KUKA KRL program: MyProgram_019().src

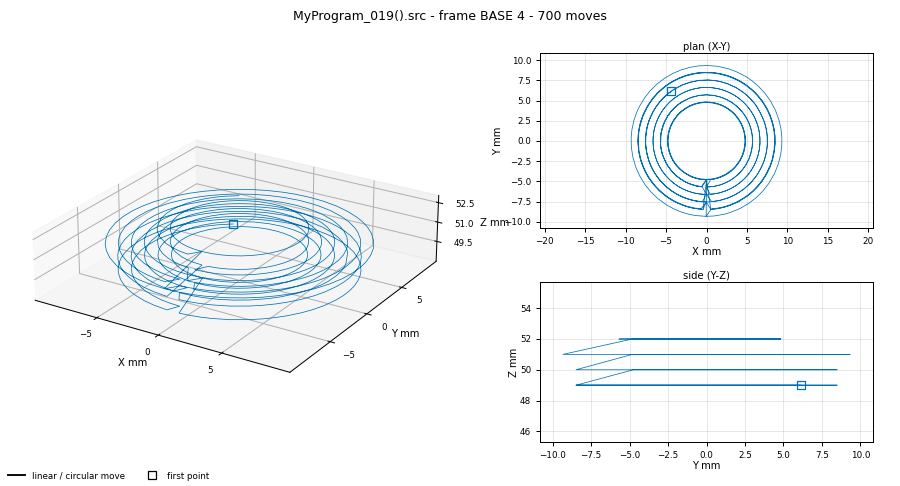
[picture p0: tool path of MyProgram_019().src in frame BASE 4, 700 of 700 moves have a stored position in this frame; points joined in program order, loops and branches not executed]
&ACCESS RVP
&REL 1
&PARAM TEMPLATE = C:\KRC\Roboter\Template\vorgabe
&PARAM EDITMASK = *
DEF MyProgram_019()
; ---- Setting reference (Base) ----
$BASE = BASE_DATA[4]

; --------------------------
; ---- Setting tool (TCP) ----
$TOOL = TOOL_DATA[3]
; --------------------------

$VEL.CP = VEL_APROX_PRINT
Startdeposition()
$VEL.CP = VEL_PRINT
LIN {X -4.3861,Y 6.1542,Z 49,A -2.5539,B 0,C 0,E1 0.1598,E2 90.072} C_DIS
LIN {X -5.2131,Y 5.4702,Z 49,A -2.6133,B 0,C 0,E1 0.1598,E2 90.0718} C_DIS
LIN {X -5.8474,Y 4.7889,Z 49,A -2.6655,B 0,C 0,E1 0.1598,E2 90.0718} C_DIS
LIN {X -6.5348,Y 3.7984,Z 49,A -2.7326,B 0,C 0,E1 0.1598,E2 90.0714} C_DIS
LIN {X -7.1278,Y 2.5114,Z 49,A -2.8086,B 0,C 0,E1 0.1598,E2 90.071} C_DIS
LIN {X -7.4027,Y 1.5183,Z 49,A -2.861,B 0,C 0,E1 0.1598,E2 90.0712} C_DIS
LIN {X -7.5273,Y 0.6846,Z 49,A -2.9011,B 0,C 0,E1 0.1598,E2 90.0714} C_DIS
LIN {X -7.5434,Y -0.4544,Z 49,A -2.9495,B 0,C 0,E1 0.1598,E2 90.0709} C_DIS
LIN {X -7.4365,Y -1.3517,Z 49,A -2.9839,B 0,C 0,E1 0.1598,E2 90.0712} C_DIS
LIN {X -7.1354,Y -2.475,Z 49,A -3.0202,B 0,C 0,E1 0.1598,E2 90.0709} C_DIS
LIN {X -6.8384,Y -3.2059,Z 49,A -3.0406,B 0,C 0,E1 0.1598,E2 90.0712} C_DIS
LIN {X -6.4681,Y -3.9026,Z 49,A -3.0566,B 0,C 0,E1 0.1598,E2 90.0712} C_DIS
LIN {X -5.8075,Y -4.8355,Z 49,A -3.0718,B 0,C 0,E1 0.1598,E2 90.071} C_DIS
LIN {X -5.1034,Y -5.5744,Z 49,A -3.0774,B 0,C 0,E1 0.1598,E2 90.0711} C_DIS
LIN {X -4.3813,Y -6.1518,Z 49,A -3.0756,B 0,C 0,E1 0.1598,E2 90.0713} C_DIS
LIN {X -3.5989,Y -6.6446,Z 49,A -3.0679,B 0,C 0,E1 0.1598,E2 90.0713} C_DIS
LIN {X -2.6446,Y -7.0747,Z 49,A -3.0512,B 0,C 0,E1 0.1598,E2 90.0713} C_DIS
LIN {X -1.6257,Y -7.3802,Z 49,A -3.0269,B 0,C 0,E1 0.1598,E2 90.0715} C_DIS
LIN {X -0.8328,Y -7.5076,Z 49,A -3.0033,B 0,C 0,E1 0.1598,E2 90.0715} C_DIS
LIN {X -0.0313,Y -7.5551,Z 49,A -2.976,B 0,C 0,E1 0.1598,E2 90.0716} C_DIS
Enddeposition()
LIN {X -0.0313,Y -7.5551,Z 49,A -2.976,B 0,C 0,E1 0.1598,E2 90.0716} C_DIS
Startdeposition()
$VEL.CP = VEL_PRINT
LIN {X -0.4344,Y -8.4805,Z 49,A -3.0298,B 0,C 0,E1 0.1598,E2 90.071} C_DIS
LIN {X -1.5865,Y -8.3368,Z 49,A -3.0665,B 0,C 0,E1 0.1598,E2 90.0714} C_DIS
LIN {X -2.5442,Y -8.1001,Z 49,A -3.0915,B 0,C 0,E1 0.1598,E2 90.0714} C_DIS
LIN {X -3.6406,Y -7.6652,Z 49,A -3.1131,B 0,C 0,E1 0.1598,E2 90.0713} C_DIS
LIN {X -4.3696,Y -7.2748,Z 49,A -3.1232,B 0,C 0,E1 0.1598,E2 90.0713} C_DIS
LIN {X -5.0572,Y -6.8153,Z 49,A -3.1289,B 0,C 0,E1 0.1598,E2 90.0713} C_DIS
LIN {X -5.8504,Y -6.1524,Z 49,A -3.1297,B 0,C 0,E1 0.1598,E2 90.0711} C_DIS
LIN {X -6.6291,Y -5.2974,Z 49,A -3.1218,B 0,C 0,E1 0.1598,E2 90.071} C_DIS
LIN {X -7.1233,Y -4.6123,Z 49,A -3.111,B 0,C 0,E1 0.1598,E2 90.0712} C_DIS
LIN {X -7.547,Y -3.8813,Z 49,A -3.0955,B 0,C 0,E1 0.1598,E2 90.0712} C_DIS
LIN {X -7.8959,Y -3.1119,Z 49,A -3.0757,B 0,C 0,E1 0.1598,E2 90.0712} C_DIS
LIN {X -8.1665,Y -2.3115,Z 49,A -3.0517,B 0,C 0,E1 0.1598,E2 90.0712} C_DIS
LIN {X -8.3936,Y -1.2801,Z 49,A -3.0161,B 0,C 0,E1 0.1598,E2 90.0709} C_DIS
LIN {X -8.487,Y -0.0694,Z 49,A -2.9681,B 0,C 0,E1 0.1598,E2 90.0709} C_DIS
LIN {X -8.4542,Y 0.7473,Z 49,A -2.9327,B 0,C 0,E1 0.1598,E2 90.0713} C_DIS
LIN {X -8.3422,Y 1.5569,Z 49,A -2.8944,B 0,C 0,E1 0.1598,E2 90.0713} C_DIS
LIN {X -8.154,Y 2.3523,Z 49,A -2.8538,B 0,C 0,E1 0.1598,E2 90.0714} C_DIS
LIN {X -7.8156,Y 3.3164,Z 49,A -2.8003,B 0,C 0,E1 0.1598,E2 90.0713} C_DIS
LIN {X -7.2981,Y 4.3333,Z 49,A -2.7381,B 0,C 0,E1 0.1598,E2 90.0713} C_DIS
LIN {X -6.6452,Y 5.2858,Z 49,A -2.6739,B 0,C 0,E1 0.1598,E2 90.0716} C_DIS
LIN {X -5.9556,Y 6.045,Z 49,A -2.6165,B 0,C 0,E1 0.1598,E2 90.0718} C_DIS
LIN {X -5.3443,Y 6.5923,Z 49,A -2.5709,B 0,C 0,E1 0.1598,E2 90.072} C_DIS
LIN {X -4.5122,Y 7.192,Z 49,A -2.5148,B 0,C 0,E1 0.1598,E2 90.072} C_DIS
LIN {X -3.4136,Y 7.7681,Z 49,A -2.4499,B 0,C 0,E1 0.1598,E2 90.0721} C_DIS
LIN {X -2.6211,Y 8.0702,Z 49,A -2.4079,B 0,C 0,E1 0.1598,E2 90.0723} C_DIS
LIN {X -1.8024,Y 8.2917,Z 49,A -2.3683,B 0,C 0,E1 0.1598,E2 90.0723} C_DIS
LIN {X -0.9657,Y 8.4308,Z 49,A -2.3315,B 0,C 0,E1 0.1598,E2 90.0725} C_DIS
LIN {X -0.1194,Y 8.4866,Z 49,A -2.2979,B 0,C 0,E1 0.1598,E2 90.0725} C_DIS
LIN {X 0.7283,Y 8.4556,Z 49,A -2.2679,B 0,C 0,E1 0.1598,E2 90.0725} C_DIS
LIN {X 1.5686,Y 8.3401,Z 49,A -2.2418,B 0,C 0,E1 0.1598,E2 90.0725} C_DIS
LIN {X 2.3934,Y 8.1418,Z 49,A -2.2198,B 0,C 0,E1 0.1598,E2 90.0725} C_DIS
LIN {X 3.1943,Y 7.8623,Z 49,A -2.2021,B 0,C 0,E1 0.1598,E2 90.0725} C_DIS
LIN {X 3.9633,Y 7.5043,Z 49,A -2.1889,B 0,C 0,E1 0.1598,E2 90.0725} C_DIS
LIN {X 4.6928,Y 7.0713,Z 49,A -2.1804,B 0,C 0,E1 0.1598,E2 90.0725} C_DIS
LIN {X 5.5399,Y 6.4335,Z 49,A -2.1761,B 0,C 0,E1 0.1598,E2 90.0724} C_DIS
LIN {X 6.4322,Y 5.5394,Z 49,A -2.1811,B 0,C 0,E1 0.1598,E2 90.0721} C_DIS
LIN {X 6.9258,Y 4.9117,Z 49,A -2.1898,B 0,C 0,E1 0.1598,E2 90.0723} C_DIS
LIN {X 7.4984,Y 3.9766,Z 49,A -2.2084,B 0,C 0,E1 0.1598,E2 90.0721} C_DIS
LIN {X 7.8686,Y 3.1812,Z 49,A -2.2288,B 0,C 0,E1 0.1598,E2 90.0722} C_DIS
LIN {X 8.1545,Y 2.3518,Z 49,A -2.2537,B 0,C 0,E1 0.1598,E2 90.0722} C_DIS
LIN {X 8.3544,Y 1.4976,Z 49,A -2.2828,B 0,C 0,E1 0.1598,E2 90.0721} C_DIS
LIN {X 8.4655,Y 0.6273,Z 49,A -2.3159,B 0,C 0,E1 0.1598,E2 90.0721} C_DIS
LIN {X 8.4847,Y -0.2497,Z 49,A -2.3526,B 0,C 0,E1 0.1598,E2 90.072} C_DIS
LIN {X 8.4122,Y -1.1239,Z 49,A -2.3927,B 0,C 0,E1 0.1598,E2 90.072} C_DIS
LIN {X 8.1761,Y -2.2938,Z 49,A -2.4511,B 0,C 0,E1 0.1598,E2 90.0716} C_DIS
LIN {X 7.8313,Y -3.2796,Z 49,A -2.506,B 0,C 0,E1 0.1598,E2 90.0716} C_DIS
LIN {X 7.4497,Y -4.0724,Z 49,A -2.5541,B 0,C 0,E1 0.1598,E2 90.0718} C_DIS
LIN {X 6.8636,Y -4.9906,Z 49,A -2.6148,B 0,C 0,E1 0.1598,E2 90.0717} C_DIS
LIN {X 6.3158,Y -5.6683,Z 49,A -2.6641,B 0,C 0,E1 0.1598,E2 90.0717} C_DIS
LIN {X 5.7013,Y -6.2863,Z 49,A -2.7131,B 0,C 0,E1 0.1598,E2 90.0717} C_DIS
LIN {X 5.0268,Y -6.8381,Z 49,A -2.7614,B 0,C 0,E1 0.1598,E2 90.0717} C_DIS
LIN {X 3.9381,Y -7.5235,Z 49,A -2.8305,B 0,C 0,E1 0.1598,E2 90.0716} C_DIS
LIN {X 2.8026,Y -8.0106,Z 49,A -2.8931,B 0,C 0,E1 0.1598,E2 90.0716} C_DIS
LIN {X 2.0583,Y -8.2323,Z 49,A -2.9299,B 0,C 0,E1 0.1598,E2 90.0716} C_DIS
LIN {X 1.2972,Y -8.386,Z 49,A -2.9643,B 0,C 0,E1 0.1598,E2 90.0716} C_DIS
LIN {X 0.5254,Y -8.4707,Z 49,A -2.9962,B 0,C 0,E1 0.1598,E2 90.0716} C_DIS
LIN {X 0.5254,Y -8.4707,Z 49,A -2.9962,B 0,C 0,E1 0.1598,E2 90.0716} C_DIS
Enddeposition()
LIN {X 0.0009,Y -4.7523,Z 50,A -2.8426,B 0,C 0,E1 0.1598,E2 90.0604} C_DIS
Startdeposition()
$VEL.CP = VEL_PRINT
LIN {X 0.0009,Y -4.7523,Z 50,A -2.8483,B 0,C 0,E1 0.1598,E2 90.0661} C_DIS
LIN {X 0.8085,Y -4.6841,Z 50,A -2.8207,B 0,C 0,E1 0.1598,E2 90.0711} C_DIS
LIN {X 1.4382,Y -4.5283,Z 50,A -2.7915,B 0,C 0,E1 0.1598,E2 90.0718} C_DIS
LIN {X 2.3301,Y -4.1421,Z 50,A -2.7423,B 0,C 0,E1 0.1598,E2 90.0718} C_DIS
LIN {X 3.1242,Y -3.5812,Z 50,A -2.6892,B 0,C 0,E1 0.1598,E2 90.0718} C_DIS
LIN {X 3.5834,Y -3.123,Z 50,A -2.6528,B 0,C 0,E1 0.1598,E2 90.0719} C_DIS
LIN {X 4.059,Y -2.467,Z 50,A -2.6072,B 0,C 0,E1 0.1598,E2 90.0719} C_DIS
LIN {X 4.4215,Y -1.7423,Z 50,A -2.5629,B 0,C 0,E1 0.1598,E2 90.0719} C_DIS
LIN {X 4.6174,Y -1.124,Z 50,A -2.5294,B 0,C 0,E1 0.1598,E2 90.0719} C_DIS
LIN {X 4.7271,Y -0.4848,Z 50,A -2.4981,B 0,C 0,E1 0.1598,E2 90.072} C_DIS
LIN {X 4.7507,Y 0.1633,Z 50,A -2.4696,B 0,C 0,E1 0.1598,E2 90.072} C_DIS
LIN {X 4.6838,Y 0.8086,Z 50,A -2.4445,B 0,C 0,E1 0.1598,E2 90.072} C_DIS
LIN {X 4.5296,Y 1.4386,Z 50,A -2.4233,B 0,C 0,E1 0.1598,E2 90.0721} C_DIS
LIN {X 4.2917,Y 2.0421,Z 50,A -2.4064,B 0,C 0,E1 0.1598,E2 90.0721} C_DIS
LIN {X 3.9731,Y 2.6071,Z 50,A -2.394,B 0,C 0,E1 0.1598,E2 90.0721} C_DIS
LIN {X 3.581,Y 3.1238,Z 50,A -2.3865,B 0,C 0,E1 0.1598,E2 90.0722} C_DIS
LIN {X 3.1226,Y 3.5827,Z 50,A -2.3839,B 0,C 0,E1 0.1598,E2 90.0722} C_DIS
LIN {X 2.6055,Y 3.9743,Z 50,A -2.3863,B 0,C 0,E1 0.1598,E2 90.0722} C_DIS
LIN {X 2.0403,Y 4.2926,Z 50,A -2.3936,B 0,C 0,E1 0.1598,E2 90.0723} C_DIS
LIN {X 1.4368,Y 4.5305,Z 50,A -2.4058,B 0,C 0,E1 0.1598,E2 90.0723} C_DIS
LIN {X 0.8065,Y 4.6839,Z 50,A -2.4225,B 0,C 0,E1 0.1598,E2 90.0723} C_DIS
LIN {X 0.1613,Y 4.7505,Z 50,A -2.4434,B 0,C 0,E1 0.1598,E2 90.0723} C_DIS
LIN {X -0.4868,Y 4.7264,Z 50,A -2.4684,B 0,C 0,E1 0.1598,E2 90.0723} C_DIS
LIN {X -1.1263,Y 4.6177,Z 50,A -2.4965,B 0,C 0,E1 0.1598,E2 90.0723} C_DIS
LIN {X -1.7444,Y 4.4207,Z 50,A -2.5277,B 0,C 0,E1 0.1598,E2 90.0722} C_DIS
LIN {X -2.3304,Y 4.1428,Z 50,A -2.561,B 0,C 0,E1 0.1598,E2 90.0722} C_DIS
LIN {X -2.8729,Y 3.7869,Z 50,A -2.5961,B 0,C 0,E1 0.1598,E2 90.072} C_DIS
LIN {X -3.3611,Y 3.3597,Z 50,A -2.6322,B 0,C 0,E1 0.1598,E2 90.072} C_DIS
LIN {X -3.7874,Y 2.8709,Z 50,A -2.6686,B 0,C 0,E1 0.1598,E2 90.0719} C_DIS
LIN {X -4.1431,Y 2.3284,Z 50,A -2.7047,B 0,C 0,E1 0.1598,E2 90.0719} C_DIS
LIN {X -4.4217,Y 1.7426,Z 50,A -2.7397,B 0,C 0,E1 0.1598,E2 90.0717} C_DIS
LIN {X -4.6178,Y 1.1244,Z 50,A -2.7732,B 0,C 0,E1 0.1598,E2 90.0717} C_DIS
LIN {X -4.7277,Y 0.4851,Z 50,A -2.8043,B 0,C 0,E1 0.1598,E2 90.0717} C_DIS
LIN {X -4.7498,Y -0.1631,Z 50,A -2.8326,B 0,C 0,E1 0.1598,E2 90.0716} C_DIS
LIN {X -4.6839,Y -0.8084,Z 50,A -2.8576,B 0,C 0,E1 0.1598,E2 90.0716} C_DIS
LIN {X -4.5298,Y -1.4385,Z 50,A -2.8787,B 0,C 0,E1 0.1598,E2 90.0716} C_DIS
LIN {X -4.2915,Y -2.0419,Z 50,A -2.8955,B 0,C 0,E1 0.1598,E2 90.0716} C_DIS
LIN {X -3.9733,Y -2.607,Z 50,A -2.9079,B 0,C 0,E1 0.1598,E2 90.0716} C_DIS
LIN {X -3.5812,Y -3.1237,Z 50,A -2.9154,B 0,C 0,E1 0.1598,E2 90.0716} C_DIS
LIN {X -3.1229,Y -3.5827,Z 50,A -2.9181,B 0,C 0,E1 0.1598,E2 90.0716} C_DIS
LIN {X -2.6057,Y -3.9741,Z 50,A -2.9158,B 0,C 0,E1 0.1598,E2 90.0716} C_DIS
LIN {X -2.0405,Y -4.2925,Z 50,A -2.9086,B 0,C 0,E1 0.1598,E2 90.0716} C_DIS
LIN {X -1.4371,Y -4.5304,Z 50,A -2.8966,B 0,C 0,E1 0.1598,E2 90.0716} C_DIS
LIN {X -0.8065,Y -4.682,Z 50,A -2.8799,B 0,C 0,E1 0.1598,E2 90.0717} C_DIS
LIN {X 0.0009,Y -4.7523,Z 50,A -2.8533,B 0,C 0,E1 0.1598,E2 90.0717} C_DIS
Enddeposition()
LIN {X 0.0009,Y -4.7523,Z 50,A -2.8533,B 0,C 0,E1 0.1598,E2 90.0717} C_DIS
Startdeposition()
$VEL.CP = VEL_PRINT
LIN {X -0.6181,Y -5.6508,Z 50,A -2.9138,B 0,C 0,E1 0.1598,E2 90.0711} C_DIS
LIN {X -1.3979,Y -5.5098,Z 50,A -2.937,B 0,C 0,E1 0.1598,E2 90.0716} C_DIS
LIN {X -2.15,Y -5.2602,Z 50,A -2.954,B 0,C 0,E1 0.1598,E2 90.0716} C_DIS
LIN {X -2.8616,Y -4.9116,Z 50,A -2.9652,B 0,C 0,E1 0.1598,E2 90.0716} C_DIS
LIN {X -3.5169,Y -4.4661,Z 50,A -2.9703,B 0,C 0,E1 0.1598,E2 90.0715} C_DIS
LIN {X -4.1036,Y -3.9332,Z 50,A -2.9691,B 0,C 0,E1 0.1598,E2 90.0715} C_DIS
LIN {X -4.6117,Y -3.3249,Z 50,A -2.9619,B 0,C 0,E1 0.1598,E2 90.0715} C_DIS
LIN {X -5.0277,Y -2.6504,Z 50,A -2.9485,B 0,C 0,E1 0.1598,E2 90.0714} C_DIS
LIN {X -5.3477,Y -1.9255,Z 50,A -2.9295,B 0,C 0,E1 0.1598,E2 90.0714} C_DIS
LIN {X -5.565,Y -1.1635,Z 50,A -2.9051,B 0,C 0,E1 0.1598,E2 90.0714} C_DIS
LIN {X -5.6725,Y -0.3782,Z 50,A -2.8757,B 0,C 0,E1 0.1598,E2 90.0714} C_DIS
LIN {X -5.607,Y 0.9677,Z 50,A -2.8155,B 0,C 0,E1 0.1598,E2 90.0708} C_DIS
LIN {X -5.2159,Y 2.259,Z 50,A -2.7466,B 0,C 0,E1 0.1598,E2 90.0711} C_DIS
LIN {X -4.8347,Y 2.9881,Z 50,A -2.7021,B 0,C 0,E1 0.1598,E2 90.0717} C_DIS
LIN {X -4.3523,Y 3.6548,Z 50,A -2.6562,B 0,C 0,E1 0.1598,E2 90.0717} C_DIS
LIN {X -3.7796,Y 4.2454,Z 50,A -2.6101,B 0,C 0,E1 0.1598,E2 90.0719} C_DIS
LIN {X -3.3003,Y 4.6348,Z 50,A -2.576,B 0,C 0,E1 0.1598,E2 90.0721} C_DIS
LIN {X -2.1072,Y 5.2844,Z 50,A -2.5044,B 0,C 0,E1 0.1598,E2 90.0721} C_DIS
LIN {X -1.0097,Y 5.6002,Z 50,A -2.4506,B 0,C 0,E1 0.1598,E2 90.0723} C_DIS
LIN {X -0.0048,Y 5.6906,Z 50,A -2.4098,B 0,C 0,E1 0.1598,E2 90.0723} C_DIS
LIN {X 1.0076,Y 5.5921,Z 50,A -2.3766,B 0,C 0,E1 0.1598,E2 90.0723} C_DIS
LIN {X 1.7959,Y 5.3908,Z 50,A -2.3561,B 0,C 0,E1 0.1598,E2 90.0723} C_DIS
LIN {X 2.5476,Y 5.0796,Z 50,A -2.3416,B 0,C 0,E1 0.1598,E2 90.0723} C_DIS
LIN {X 3.2472,Y 4.6641,Z 50,A -2.3334,B 0,C 0,E1 0.1598,E2 90.0723} C_DIS
LIN {X 3.8795,Y 4.1521,Z 50,A -2.3319,B 0,C 0,E1 0.1598,E2 90.0723} C_DIS
LIN {X 4.4334,Y 3.5562,Z 50,A -2.3368,B 0,C 0,E1 0.1598,E2 90.0723} C_DIS
LIN {X 4.8952,Y 2.8862,Z 50,A -2.3483,B 0,C 0,E1 0.1598,E2 90.0722} C_DIS
LIN {X 5.2572,Y 2.1576,Z 50,A -2.366,B 0,C 0,E1 0.1598,E2 90.0721} C_DIS
LIN {X 5.5127,Y 1.385,Z 50,A -2.3895,B 0,C 0,E1 0.1598,E2 90.0721} C_DIS
LIN {X 5.6553,Y 0.5837,Z 50,A -2.4184,B 0,C 0,E1 0.1598,E2 90.072} C_DIS
LIN {X 5.6811,Y -0.2299,Z 50,A -2.4521,B 0,C 0,E1 0.1598,E2 90.072} C_DIS
LIN {X 5.5897,Y -1.0387,Z 50,A -2.49,B 0,C 0,E1 0.1598,E2 90.0719} C_DIS
LIN {X 5.2795,Y -2.123,Z 50,A -2.5475,B 0,C 0,E1 0.1598,E2 90.0716} C_DIS
LIN {X 4.8774,Y -2.919,Z 50,A -2.5965,B 0,C 0,E1 0.1598,E2 90.0718} C_DIS
LIN {X 4.4734,Y -3.5068,Z 50,A -2.6366,B 0,C 0,E1 0.1598,E2 90.0718} C_DIS
LIN {X 3.9995,Y -4.0396,Z 50,A -2.6767,B 0,C 0,E1 0.1598,E2 90.0718} C_DIS
LIN {X 3.4612,Y -4.5075,Z 50,A -2.7165,B 0,C 0,E1 0.1598,E2 90.0718} C_DIS
LIN {X 2.8706,Y -4.9075,Z 50,A -2.7553,B 0,C 0,E1 0.1598,E2 90.0718} C_DIS
LIN {X 2.2325,Y -5.2263,Z 50,A -2.7923,B 0,C 0,E1 0.1598,E2 90.0718} C_DIS
LIN {X 1.5614,Y -5.468,Z 50,A -2.8273,B 0,C 0,E1 0.1598,E2 90.0718} C_DIS
LIN {X 0.8645,Y -5.6203,Z 50,A -2.8593,B 0,C 0,E1 0.1598,E2 90.0718} C_DIS
LIN {X -0.0245,Y -5.6887,Z 50,A -2.8949,B 0,C 0,E1 0.1598,E2 90.0718} C_DIS
Enddeposition()
LIN {X -0.0245,Y -5.6887,Z 50,A -2.8949,B 0,C 0,E1 0.1598,E2 90.0718} C_DIS
Startdeposition()
$VEL.CP = VEL_PRINT
LIN {X 0.471,Y -6.6032,Z 50,A -2.4861,B -0.0002,C -0.0012,E1 0.1597,E2 89.6399} C_DIS
LIN {X 1.1476,Y -6.5205,Z 50,A -2.4647,B -0.0002,C -0.0012,E1 0.1596,E2 89.6469} C_DIS
LIN {X 1.812,Y -6.3679,Z 50,A -2.4453,B -0.0004,C -0.0012,E1 0.1594,E2 89.6583} C_DIS
LIN {X 2.4566,Y -6.1466,Z 50,A -2.427,B -0.0005,C -0.0011,E1 0.1594,E2 89.6731} C_DIS
LIN {X 3.0753,Y -5.8607,Z 50,A -2.4114,B -0.0006,C -0.0011,E1 0.1592,E2 89.6924} C_DIS
LIN {X 3.6623,Y -5.5143,Z 50,A -2.3987,B -0.0007,C -0.001,E1 0.1591,E2 89.7161} C_DIS
LIN {X 4.2103,Y -5.1088,Z 50,A -2.3891,B -0.0008,C -0.0009,E1 0.159,E2 89.7442} C_DIS
LIN {X 4.713,Y -4.6485,Z 50,A -2.3807,B -0.0009,C -0.0008,E1 0.159,E2 89.7741} C_DIS
LIN {X 5.1664,Y -4.1397,Z 50,A -2.3773,B -0.0009,C -0.0007,E1 0.1588,E2 89.8094} C_DIS
LIN {X 5.5644,Y -3.5864,Z 50,A -2.3753,B -0.0011,C -0.0006,E1 0.1588,E2 89.8459} C_DIS
LIN {X 5.9027,Y -2.9948,Z 50,A -2.3772,B -0.0011,C -0.0005,E1 0.1587,E2 89.8859} C_DIS
LIN {X 6.1796,Y -2.372,Z 50,A -2.3813,B -0.0011,C -0.0004,E1 0.1587,E2 89.9271} C_DIS
LIN {X 6.3904,Y -1.7239,Z 50,A -2.389,B -0.0011,C -0.0002,E1 0.1587,E2 89.9706} C_DIS
LIN {X 6.5347,Y -1.0577,Z 50,A -2.3962,B -0.0012,C -0.0002,E1 0.1586,E2 90.0119} C_DIS
LIN {X 6.6093,Y -0.3803,Z 50,A -2.4142,B -0.0012,C 0,E1 0.1586,E2 90.0619} C_DIS
LIN {X 6.6111,Y 0.3014,Z 50,A -2.4244,B -0.0012,C 0.0001,E1 0.1586,E2 90.1015} C_DIS
LIN {X 6.5462,Y 0.9798,Z 50,A -2.4456,B -0.0012,C 0.0003,E1 0.1586,E2 90.1495} C_DIS
LIN {X 6.4118,Y 1.6481,Z 50,A -2.4626,B -0.0012,C 0.0003,E1 0.1586,E2 90.1902} C_DIS
LIN {X 6.2105,Y 2.2993,Z 50,A -2.487,B -0.0012,C 0.0005,E1 0.1586,E2 90.2351} C_DIS
LIN {X 5.9408,Y 2.9254,Z 50,A -2.5107,B -0.001,C 0.0006,E1 0.1587,E2 90.2756} C_DIS
LIN {X 5.6083,Y 3.5204,Z 50,A -2.5361,B -0.001,C 0.0007,E1 0.1587,E2 90.314} C_DIS
LIN {X 5.2166,Y 4.0784,Z 50,A -2.5627,B -0.0009,C 0.0008,E1 0.1589,E2 90.3499} C_DIS
LIN {X 4.7691,Y 4.5926,Z 50,A -2.5902,B -0.0009,C 0.0008,E1 0.1589,E2 90.3827} C_DIS
LIN {X 4.2721,Y 5.0593,Z 50,A -2.6185,B -0.0007,C 0.001,E1 0.159,E2 90.4123} C_DIS
LIN {X 3.7285,Y 5.4706,Z 50,A -2.6478,B -0.0007,C 0.001,E1 0.1591,E2 90.4388} C_DIS
LIN {X 3.1458,Y 5.8244,Z 50,A -2.6759,B -0.0005,C 0.0011,E1 0.1592,E2 90.4601} C_DIS
LIN {X 2.5307,Y 6.1182,Z 50,A -2.704,B -0.0004,C 0.0011,E1 0.1594,E2 90.4778} C_DIS
LIN {X 1.8883,Y 6.346,Z 50,A -2.7323,B -0.0003,C 0.0011,E1 0.1594,E2 90.4917} C_DIS
LIN {X 1.2257,Y 6.5057,Z 50,A -2.759,B -0.0001,C 0.0012,E1 0.1596,E2 90.5005} C_DIS
LIN {X 0.5501,Y 6.5957,Z 50,A -2.7848,B -0.0001,C 0.0012,E1 0.1597,E2 90.5049} C_DIS
LIN {X -0.1312,Y 6.6187,Z 50,A -2.8092,B 0.0001,C 0.0012,E1 0.1598,E2 90.5049} C_DIS
LIN {X -0.8111,Y 6.5716,Z 50,A -2.8316,B 0.0002,C 0.0012,E1 0.16,E2 90.4998} C_DIS
LIN {X -1.4822,Y 6.4525,Z 50,A -2.8521,B 0.0004,C 0.0012,E1 0.16,E2 90.4903} C_DIS
LIN {X -2.1375,Y 6.265,Z 50,A -2.8713,B 0.0004,C 0.0012,E1 0.1602,E2 90.4773} C_DIS
LIN {X -2.7706,Y 6.0125,Z 50,A -2.8871,B 0.0006,C 0.0011,E1 0.1603,E2 90.459} C_DIS
LIN {X -3.374,Y 5.6956,Z 50,A -2.9008,B 0.0006,C 0.001,E1 0.1604,E2 90.4369} C_DIS
LIN {X -3.9417,Y 5.3185,Z 50,A -2.9118,B 0.0008,C 0.001,E1 0.1605,E2 90.4111} C_DIS
LIN {X -4.4677,Y 4.885,Z 50,A -2.9192,B 0.0008,C 0.0008,E1 0.1606,E2 90.3808} C_DIS
LIN {X -4.9453,Y 4.3989,Z 50,A -2.9259,B 0.001,C 0.0008,E1 0.1607,E2 90.3494} C_DIS
LIN {X -5.3717,Y 3.8672,Z 50,A -2.9292,B 0.001,C 0.0006,E1 0.1607,E2 90.3146} C_DIS
LIN {X -5.742,Y 3.2949,Z 50,A -2.9276,B 0.001,C 0.0006,E1 0.1609,E2 90.2753} C_DIS
LIN {X -6.0503,Y 2.6871,Z 50,A -2.9252,B 0.0011,C 0.0004,E1 0.1609,E2 90.236} C_DIS
LIN {X -6.2956,Y 2.0512,Z 50,A -2.9188,B 0.0011,C 0.0003,E1 0.1609,E2 90.1939} C_DIS
LIN {X -6.4739,Y 1.3932,Z 50,A -2.91,B 0.0011,C 0.0002,E1 0.1609,E2 90.1509} C_DIS
LIN {X -6.5829,Y 0.7203,Z 50,A -2.8973,B 0.0012,C 0,E1 0.1609,E2 90.1058} C_DIS
LIN {X -6.6203,Y 0.0397,Z 50,A -2.8828,B 0.0012,C 0,E1 0.1609,E2 90.0614} C_DIS
LIN {X -6.5889,Y -0.6412,Z 50,A -2.8682,B 0.0012,C -0.0002,E1 0.1609,E2 90.0192} C_DIS
LIN {X -6.4899,Y -1.3156,Z 50,A -2.8489,B 0.0012,C -0.0003,E1 0.1609,E2 89.9751} C_DIS
LIN {X -6.3209,Y -1.976,Z 50,A -2.8273,B 0.0012,C -0.0004,E1 0.1609,E2 89.9318} C_DIS
LIN {X -6.0839,Y -2.6152,Z 50,A -2.8045,B 0.0011,C -0.0006,E1 0.1609,E2 89.8906} C_DIS
LIN {X -5.7823,Y -3.2265,Z 50,A -2.779,B 0.0011,C -0.0006,E1 0.1609,E2 89.8502} C_DIS
LIN {X -5.4183,Y -3.803,Z 50,A -2.7553,B 0.0009,C -0.0008,E1 0.1608,E2 89.8152} C_DIS
LIN {X -4.9996,Y -4.3409,Z 50,A -2.7285,B 0.0009,C -0.0008,E1 0.1607,E2 89.7809} C_DIS
LIN {X -4.5271,Y -4.8321,Z 50,A -2.699,B 0.0008,C -0.0009,E1 0.1606,E2 89.7477} C_DIS
LIN {X -4.0043,Y -5.2695,Z 50,A -2.6723,B 0.0007,C -0.001,E1 0.1605,E2 89.7214} C_DIS
LIN {X -3.4417,Y -5.6543,Z 50,A -2.6437,B 0.0006,C -0.001,E1 0.1604,E2 89.6969} C_DIS
LIN {X -2.8419,Y -5.9783,Z 50,A -2.6165,B 0.0004,C -0.0011,E1 0.1603,E2 89.6776} C_DIS
LIN {X -2.2129,Y -6.2406,Z 50,A -2.5878,B 0.0004,C -0.0011,E1 0.1602,E2 89.6606} C_DIS
LIN {X -1.5595,Y -6.4344,Z 50,A -2.5606,B 0.0002,C -0.0011,E1 0.16,E2 89.6488} C_DIS
LIN {X -0.8897,Y -6.561,Z 50,A -2.5344,B 0.0001,C -0.0012,E1 0.16,E2 89.6416} C_DIS
LIN {X -0.0401,Y -6.6227,Z 50,A -2.5035,B 0,C -0.0012,E1 0.1598,E2 89.639} C_DIS
Enddeposition()
LIN {X -0.0401,Y -6.6227,Z 50,A -2.5035,B 0,C -0.0012,E1 0.1598,E2 89.639} C_DIS
Startdeposition()
$VEL.CP = VEL_PRINT
LIN {X -0.51,Y -7.5373,Z 50,A -2.4184,B 0,C -0.0016,E1 0.1599,E2 89.4966} C_DIS
LIN {X -1.1463,Y -7.465,Z 50,A -2.4452,B 0.0002,C -0.0016,E1 0.1601,E2 89.5035} C_DIS
LIN {X -2.151,Y -7.2449,Z 50,A -2.4933,B 0.0004,C -0.0016,E1 0.1603,E2 89.5247} C_DIS
LIN {X -3.1222,Y -6.8837,Z 50,A -2.5456,B 0.0007,C -0.0015,E1 0.1605,E2 89.5572} C_DIS
LIN {X -4.0717,Y -6.3617,Z 50,A -2.5961,B 0.0008,C -0.0014,E1 0.1607,E2 89.5956} C_DIS
LIN {X -4.6767,Y -5.9319,Z 50,A -2.632,B 0.001,C -0.0013,E1 0.1608,E2 89.6279} C_DIS
LIN {X -5.5156,Y -5.1654,Z 50,A -2.6931,B 0.0012,C -0.0011,E1 0.161,E2 89.6912} C_DIS
LIN {X -6.1426,Y -4.4029,Z 50,A -2.7427,B 0.0012,C -0.001,E1 0.1611,E2 89.7504} C_DIS
LIN {X -6.6609,Y -3.5627,Z 50,A -2.7909,B 0.0014,C -0.0008,E1 0.1612,E2 89.8154} C_DIS
LIN {X -6.9946,Y -2.847,Z 50,A -2.8253,B 0.0014,C -0.0006,E1 0.1612,E2 89.8679} C_DIS
LIN {X -7.3109,Y -1.912,Z 50,A -2.8747,B 0.0016,C -0.0004,E1 0.1614,E2 89.9452} C_DIS
LIN {X -7.5223,Y -0.6826,Z 50,A -2.9028,B 0.0016,C -0.0002,E1 0.1614,E2 90.0174} C_DIS
LIN {X -7.555,Y 0.1746,Z 50,A -2.9521,B 0.0016,C 0,E1 0.1614,E2 90.1014} C_DIS
LIN {X -7.4392,Y 1.3106,Z 50,A -2.9676,B 0.0016,C 0.0002,E1 0.1614,E2 90.169} C_DIS
LIN {X -7.2716,Y 2.0585,Z 50,A -3.0047,B 0.0016,C 0.0004,E1 0.1614,E2 90.2435} C_DIS
LIN {X -6.8991,Y 3.0831,Z 50,A -3.035,B 0.0015,C 0.0007,E1 0.1612,E2 90.3303} C_DIS
LIN {X -6.2055,Y 4.3037,Z 50,A -3.0358,B 0.0014,C 0.0009,E1 0.1612,E2 90.4078} C_DIS
LIN {X -5.4947,Y 5.1873,Z 50,A -3.0401,B 0.0012,C 0.0011,E1 0.1609,E2 90.4753} C_DIS
LIN {X -4.7594,Y 5.8717,Z 50,A -3.0376,B 0.001,C 0.0012,E1 0.1608,E2 90.5288} C_DIS
LIN {X -3.9242,Y 6.4579,Z 50,A -3.0262,B 0.0009,C 0.0014,E1 0.1606,E2 90.5729} C_DIS
LIN {X -3.0346,Y 6.921,Z 50,A -3.008,B 0.0007,C 0.0014,E1 0.1604,E2 90.6072} C_DIS
LIN {X -2.1174,Y 7.2554,Z 50,A -2.9828,B 0.0005,C 0.0015,E1 0.1602,E2 90.6302} C_DIS
LIN {X -0.9577,Y 7.4967,Z 50,A -2.9454,B 0.0002,C 0.0015,E1 0.16,E2 90.6463} C_DIS
LIN {X 0.3556,Y 7.5501,Z 50,A -2.8959,B -0.0001,C 0.0016,E1 0.1597,E2 90.6482} C_DIS
LIN {X 1.4005,Y 7.4275,Z 50,A -2.8515,B -0.0003,C 0.0016,E1 0.1595,E2 90.6377} C_DIS
LIN {X 2.5747,Y 7.1046,Z 50,A -2.794,B -0.0005,C 0.0016,E1 0.1592,E2 90.6107} C_DIS
LIN {X 3.6494,Y 6.6125,Z 50,A -2.7358,B -0.0008,C 0.0014,E1 0.159,E2 90.5719} C_DIS
LIN {X 4.3896,Y 6.145,Z 50,A -2.6921,B -0.0009,C 0.0014,E1 0.1588,E2 90.536} C_DIS
LIN {X 5.072,Y 5.5966,Z 50,A -2.6466,B -0.0011,C 0.0012,E1 0.1587,E2 90.4928} C_DIS
LIN {X 5.8746,Y 4.7562,Z 50,A -2.5818,B -0.0012,C 0.001,E1 0.1585,E2 90.4222} C_DIS
LIN {X 6.2921,Y 4.1866,Z 50,A -2.5309,B -0.0014,C 0.0009,E1 0.1584,E2 90.3625} C_DIS
LIN {X 7.2019,Y 2.2885,Z 50,A -2.4486,B -0.0015,C 0.0005,E1 0.1582,E2 90.2328} C_DIS
LIN {X 7.438,Y 1.3426,Z 50,A -2.4046,B -0.0015,C 0.0003,E1 0.1582,E2 90.1568} C_DIS
LIN {X 7.5467,Y 0.4057,Z 50,A -2.3682,B -0.0016,C 0.0001,E1 0.1582,E2 90.084} C_DIS
LIN {X 7.5248,Y -0.67,Z 50,A -2.338,B -0.0016,C -0.0001,E1 0.1582,E2 90.0065} C_DIS
LIN {X 7.4207,Y -1.4151,Z 50,A -2.3173,B -0.0016,C -0.0003,E1 0.1582,E2 89.9497} C_DIS
LIN {X 7.1523,Y -2.4446,Z 50,A -2.289,B -0.0016,C -0.0005,E1 0.1582,E2 89.8668} C_DIS
LIN {X 6.7592,Y -3.3699,Z 50,A -2.2776,B -0.0015,C -0.0007,E1 0.1584,E2 89.8008} C_DIS
LIN {X 6.0895,Y -4.4773,Z 50,A -2.2666,B -0.0013,C -0.0009,E1 0.1585,E2 89.7171} C_DIS
LIN {X 5.5264,Y -5.1539,Z 50,A -2.2644,B -0.0012,C -0.0011,E1 0.1586,E2 89.6649} C_DIS
LIN {X 4.5596,Y -6.0261,Z 50,A -2.2714,B -0.001,C -0.0013,E1 0.1589,E2 89.5986} C_DIS
LIN {X 3.6748,Y -6.6029,Z 50,A -2.2869,B -0.0008,C -0.0014,E1 0.1591,E2 89.5568} C_DIS
LIN {X 2.7499,Y -7.0401,Z 50,A -2.3095,B -0.0006,C -0.0014,E1 0.1593,E2 89.5267} C_DIS
LIN {X 1.7807,Y -7.3403,Z 50,A -2.3372,B -0.0004,C -0.0016,E1 0.1595,E2 89.5062} C_DIS
LIN {X 0.9826,Y -7.4892,Z 50,A -2.3637,B -0.0002,C -0.0016,E1 0.1596,E2 89.4971} C_DIS
LIN {X -0.0298,Y -7.5552,Z 50,A -2.4005,B -0.0001,C -0.0016,E1 0.1598,E2 89.4944} C_DIS
Enddeposition()
LIN {X -0.0298,Y -7.5552,Z 50,A -2.4005,B -0.0001,C -0.0016,E1 0.1598,E2 89.4944} C_DIS
Startdeposition()
$VEL.CP = VEL_PRINT
LIN {X 0.528,Y -8.4707,Z 50,A -2.2576,B -0.0003,C -0.0021,E1 0.1596,E2 89.3312} C_DIS
LIN {X 1.2997,Y -8.3857,Z 50,A -2.2346,B -0.0004,C -0.0021,E1 0.1594,E2 89.3398} C_DIS
LIN {X 2.0606,Y -8.2318,Z 50,A -2.2145,B -0.0006,C -0.002,E1 0.1593,E2 89.354} C_DIS
LIN {X 2.8046,Y -8.01,Z 50,A -2.1978,B -0.0008,C -0.002,E1 0.1591,E2 89.374} C_DIS
LIN {X 3.9381,Y -7.5236,Z 50,A -2.1865,B -0.0011,C -0.0018,E1 0.1588,E2 89.4252} C_DIS
LIN {X 5.0367,Y -6.8306,Z 50,A -2.1737,B -0.0013,C -0.0016,E1 0.1585,E2 89.4826} C_DIS
LIN {X 5.7197,Y -6.269,Z 50,A -2.1749,B -0.0015,C -0.0014,E1 0.1584,E2 89.5332} C_DIS
LIN {X 6.3406,Y -5.6395,Z 50,A -2.1812,B -0.0016,C -0.0013,E1 0.1582,E2 89.5897} C_DIS
LIN {X 6.8925,Y -4.9489,Z 50,A -2.192,B -0.0018,C -0.0011,E1 0.1581,E2 89.651} C_DIS
LIN {X 7.3711,Y -4.2054,Z 50,A -2.2079,B -0.0018,C -0.0009,E1 0.158,E2 89.7168} C_DIS
LIN {X 7.8827,Y -3.1588,Z 50,A -2.2384,B -0.002,C -0.0006,E1 0.1579,E2 89.8119} C_DIS
LIN {X 8.1753,Y -2.2973,Z 50,A -2.2733,B -0.002,C -0.0004,E1 0.1578,E2 89.8952} C_DIS
LIN {X 8.4139,Y -1.1128,Z 50,A -2.3105,B -0.002,C -0.0001,E1 0.1578,E2 89.9927} C_DIS
LIN {X 8.4857,Y -0.2323,Z 50,A -2.3487,B -0.002,C 0.0001,E1 0.1578,E2 90.0718} C_DIS
LIN {X 8.4633,Y 0.6508,Z 50,A -2.3912,B -0.002,C 0.0003,E1 0.1578,E2 90.1518} C_DIS
LIN {X 8.3485,Y 1.5268,Z 50,A -2.4341,B -0.002,C 0.0005,E1 0.1578,E2 90.2282} C_DIS
LIN {X 8.1438,Y 2.3861,Z 50,A -2.4791,B -0.002,C 0.0007,E1 0.1578,E2 90.3027} C_DIS
LIN {X 7.8524,Y 3.2201,Z 50,A -2.5275,B -0.0019,C 0.0009,E1 0.1578,E2 90.3761} C_DIS
LIN {X 7.4752,Y 4.019,Z 50,A -2.5757,B -0.0018,C 0.0011,E1 0.158,E2 90.4445} C_DIS
LIN {X 6.8558,Y 5.0116,Z 50,A -2.6441,B -0.0016,C 0.0013,E1 0.1582,E2 90.5321} C_DIS
LIN {X 5.9816,Y 6.0279,Z 50,A -2.7259,B -0.0013,C 0.0016,E1 0.1584,E2 90.6245} C_DIS
LIN {X 5.0282,Y 6.8376,Z 50,A -2.7893,B -0.0011,C 0.0018,E1 0.1586,E2 90.6865} C_DIS
LIN {X 4.3078,Y 7.3127,Z 50,A -2.8355,B -0.0009,C 0.0018,E1 0.1588,E2 90.7257} C_DIS
LIN {X 3.543,Y 7.7125,Z 50,A -2.88,B -0.0007,C 0.0019,E1 0.159,E2 90.7583} C_DIS
LIN {X 2.7415,Y 8.0326,Z 50,A -2.9219,B -0.0005,C 0.002,E1 0.1592,E2 90.7836} C_DIS
LIN {X 1.9117,Y 8.2696,Z 50,A -2.9611,B -0.0003,C 0.002,E1 0.1594,E2 90.8015} C_DIS
LIN {X 1.0621,Y 8.4213,Z 50,A -2.9969,B -0.0001,C 0.002,E1 0.1596,E2 90.8117} C_DIS
LIN {X 0.2016,Y 8.4866,Z 50,A -3.0291,B 0.0001,C 0.002,E1 0.1598,E2 90.8144} C_DIS
LIN {X -0.661,Y 8.4626,Z 50,A -3.0573,B 0.0003,C 0.002,E1 0.16,E2 90.8092} C_DIS
LIN {X -1.5168,Y 8.3511,Z 50,A -3.0814,B 0.0005,C 0.002,E1 0.1602,E2 90.7966} C_DIS
LIN {X -2.357,Y 8.1538,Z 50,A -3.101,B 0.0007,C 0.002,E1 0.1604,E2 90.7765} C_DIS
LIN {X -3.1728,Y 7.8723,Z 50,A -3.1159,B 0.0009,C 0.0019,E1 0.1606,E2 90.7491} C_DIS
LIN {X -4.1469,Y 7.4088,Z 50,A -3.124,B 0.0012,C 0.0017,E1 0.1609,E2 90.7015} C_DIS
LIN {X -5.0415,Y 6.8334,Z 50,A -3.1246,B 0.0014,C 0.0015,E1 0.1611,E2 90.6449} C_DIS
LIN {X -5.9848,Y 6.0174,Z 50,A -3.129,B 0.0016,C 0.0014,E1 0.1613,E2 90.5803} C_DIS
LIN {X -6.6453,Y 5.2858,Z 50,A -3.1124,B 0.0017,C 0.0011,E1 0.1615,E2 90.5089} C_DIS
LIN {X -7.3008,Y 4.3288,Z 50,A -3.0966,B 0.0019,C 0.0009,E1 0.1616,E2 90.429} C_DIS
LIN {X -7.8181,Y 3.3108,Z 50,A -3.0679,B 0.0019,C 0.0007,E1 0.1617,E2 90.3388} C_DIS
LIN {X -8.1738,Y 2.3031,Z 50,A -3.0339,B 0.002,C 0.0004,E1 0.1618,E2 90.2498} C_DIS
LIN {X -8.396,Y 1.2405,Z 50,A -2.9953,B 0.002,C 0.0001,E1 0.1618,E2 90.1587} C_DIS
LIN {X -8.4923,Y 0.0107,Z 50,A -2.9427,B 0.002,C -0.0002,E1 0.1618,E2 90.0512} C_DIS
LIN {X -8.3936,Y -1.281,Z 50,A -2.883,B 0.002,C -0.0005,E1 0.1618,E2 89.9409} C_DIS
LIN {X -8.1664,Y -2.3122,Z 50,A -2.8296,B 0.002,C -0.0007,E1 0.1618,E2 89.8524} C_DIS
LIN {X -7.8958,Y -3.1124,Z 50,A -2.7851,B 0.0019,C -0.0009,E1 0.1617,E2 89.784} C_DIS
LIN {X -7.5468,Y -3.8817,Z 50,A -2.7389,B 0.0018,C -0.0011,E1 0.1617,E2 89.718} C_DIS
LIN {X -7.1232,Y -4.6125,Z 50,A -2.6922,B 0.0017,C -0.0012,E1 0.1615,E2 89.6557} C_DIS
LIN {X -6.6291,Y -5.2975,Z 50,A -2.6465,B 0.0015,C -0.0014,E1 0.1614,E2 89.5989} C_DIS
LIN {X -5.8475,Y -6.1554,Z 50,A -2.5802,B 0.0013,C -0.0016,E1 0.1612,E2 89.5244} C_DIS
LIN {X -5.054,Y -6.8178,Z 50,A -2.5235,B 0.0011,C -0.0017,E1 0.161,E2 89.4681} C_DIS
LIN {X -4.3662,Y -7.2768,Z 50,A -2.4795,B 0.0009,C -0.0018,E1 0.1608,E2 89.4293} C_DIS
LIN {X -3.6372,Y -7.6668,Z 50,A -2.4383,B 0.0008,C -0.0019,E1 0.1606,E2 89.3977} C_DIS
LIN {X -2.5379,Y -8.1022,Z 50,A -2.3798,B 0.0005,C -0.002,E1 0.1604,E2 89.3602} C_DIS
LIN {X -1.5825,Y -8.3377,Z 50,A -2.3364,B 0.0003,C -0.002,E1 0.1601,E2 89.3412} C_DIS
LIN {X -0.4265,Y -8.4811,Z 50,A -2.2898,B 0,C -0.002,E1 0.1599,E2 89.3301} C_DIS
LIN {X -0.4265,Y -8.4811,Z 50,A -2.2898,B 0,C -0.002,E1 0.1599,E2 89.3301} C_DIS
Enddeposition()
LIN {X 0.0026,Y -4.8185,Z 51,A -84.6758,B 0.9069,C 0.118,E1 0.9225,E2 172.1056} C_DIS
Startdeposition()
$VEL.CP = VEL_PRINT
LIN {X -0.7076,Y -4.7624,Z 51,A -92.7843,B 0.9067,C 0.1196,E1 0.8997,E2 180.2162} C_DIS
LIN {X -1.2653,Y -4.6447,Z 51,A -99.4873,B 0.9068,C 0.1185,E1 0.8812,E2 186.9216} C_DIS
LIN {X -1.9385,Y -4.4113,Z 51,A -109.7763,B 0.9076,C 0.1126,E1 0.8541,E2 197.2219} C_DIS
LIN {X -2.8365,Y -3.8866,Z 51,A -121.9743,B 0.9092,C 0.0991,E1 0.8251,E2 209.4227} C_DIS
LIN {X -3.3473,Y -3.4577,Z 51,A -130.434,B 0.9105,C 0.086,E1 0.8074,E2 217.8864} C_DIS
LIN {X -3.7937,Y -2.962,Z 51,A -139.7233,B 0.912,C 0.0685,E1 0.7905,E2 227.1826} C_DIS
LIN {X -4.1681,Y -2.4097,Z 51,A -149.2106,B 0.9133,C 0.0477,E1 0.7764,E2 236.6768} C_DIS
LIN {X -4.4589,Y -1.8093,Z 51,A -158.0083,B 0.9142,C 0.0262,E1 0.7664,E2 245.478} C_DIS
LIN {X -4.6677,Y -1.1757,Z 51,A -167.8764,B 0.9146,C 0.0003,E1 0.7587,E2 255.353} C_DIS
LIN {X -4.7861,Y -0.5192,Z 51,A -177.3655,B 0.9142,C -0.0257,E1 0.7549,E2 264.8468} C_DIS
LIN {X -4.8115,Y 0.1475,Z 51,A 172.8273,B 0.913,C -0.053,E1 0.7548,E2 274.659} C_DIS
LIN {X -4.7445,Y 0.8112,Z 51,A 163.497,B 0.9112,C -0.0786,E1 0.7583,E2 283.9921} C_DIS
LIN {X -4.5878,Y 1.4597,Z 51,A 153.9122,B 0.9086,C -0.1037,E1 0.7654,E2 293.58} C_DIS
LIN {X -4.3408,Y 2.0793,Z 51,A 144.362,B 0.9057,C -0.127,E1 0.7761,E2 303.1323} C_DIS
LIN {X -4.0125,Y 2.6602,Z 51,A 135.1943,B 0.9026,C -0.1471,E1 0.7896,E2 312.3007} C_DIS
LIN {X -3.6059,Y 3.1891,Z 51,A 126.1158,B 0.8997,C -0.1644,E1 0.8059,E2 321.3792} C_DIS
LIN {X -3.1301,Y 3.6569,Z 51,A 117.141,B 0.897,C -0.1783,E1 0.8245,E2 330.3533} C_DIS
LIN {X -2.5933,Y 4.0529,Z 51,A 108.9555,B 0.895,C -0.1881,E1 0.8436,E2 338.5359} C_DIS
LIN {X -2.0087,Y 4.374,Z 51,A 100.2378,B 0.8935,C -0.1952,E1 0.8656,E2 347.2521} C_DIS
LIN {X -1.3847,Y 4.6098,Z 51,A 92.3222,B 0.8927,C -0.1986,E1 0.8868,E2 355.164} C_DIS
LIN {X -0.7342,Y 4.7576,Z 51,A 84.249,B 0.8927,C -0.199,E1 0.9093,E2 363.2339} C_DIS
LIN {X -0.0694,Y 4.8129,Z 51,A 76.4191,B 0.8932,C -0.1964,E1 0.9314,E2 371.06} C_DIS
LIN {X 0.5966,Y 4.7764,Z 51,A 68.7476,B 0.8944,C -0.191,E1 0.953,E2 378.7275} C_DIS
LIN {X 1.2512,Y 4.6477,Z 51,A 61.3258,B 0.896,C -0.1832,E1 0.9735,E2 386.1449} C_DIS
LIN {X 1.881,Y 4.4284,Z 51,A 54.2108,B 0.8979,C -0.1735,E1 0.9922,E2 393.2548} C_DIS
LIN {X 2.477,Y 4.1286,Z 51,A 46.8142,B 0.9002,C -0.1613,E1 1.0104,E2 400.6476} C_DIS
LIN {X 3.0221,Y 3.744,Z 51,A 39.7205,B 0.9026,C -0.1477,E1 1.0264,E2 407.7366} C_DIS
LIN {X 3.5119,Y 3.2912,Z 51,A 32.9198,B 0.9048,C -0.1331,E1 1.0399,E2 414.5325} C_DIS
LIN {X 3.933,Y 2.774,Z 51,A 25.8928,B 0.9071,C -0.1166,E1 1.0518,E2 421.5555} C_DIS
LIN {X 4.279,Y 2.2037,Z 51,A 19.0214,B 0.9091,C -0.0994,E1 1.0612,E2 428.4228} C_DIS
LIN {X 4.5426,Y 1.5909,Z 51,A 12.2223,B 0.9109,C -0.0815,E1 1.0681,E2 435.218} C_DIS
LIN {X 4.7192,Y 0.9477,Z 51,A 5.4456,B 0.9124,C -0.063,E1 1.0725,E2 441.991} C_DIS
LIN {X 4.8052,Y 0.2862,Z 51,A -1.1801,B 0.9135,C -0.0447,E1 1.0743,E2 448.6128} C_DIS
LIN {X 4.8001,Y -0.3809,Z 51,A -8.1044,B 0.9142,C -0.0255,E1 1.0735,E2 455.5349} C_DIS
LIN {X 4.7018,Y -1.041,Z 51,A -15.0492,B 0.9145,C -0.0064,E1 1.0699,E2 462.4777} C_DIS
LIN {X 4.5118,Y -1.6807,Z 51,A -21.9244,B 0.9145,C 0.0121,E1 1.0638,E2 469.351} C_DIS
LIN {X 4.2339,Y -2.2871,Z 51,A -28.2908,B 0.9141,C 0.0285,E1 1.0559,E2 475.7136} C_DIS
LIN {X 3.8782,Y -2.8515,Z 51,A -35.6514,B 0.9134,C 0.0464,E1 1.0443,E2 483.075} C_DIS
LIN {X 3.4459,Y -3.3597,Z 51,A -42.1272,B 0.9125,C 0.061,E1 1.032,E2 489.5479} C_DIS
LIN {X 2.95,Y -3.806,Z 51,A -49.5599,B 0.9114,C 0.0762,E1 1.016,E2 496.9822} C_DIS
LIN {X 2.3951,Y -4.1765,Z 51,A -56.7192,B 0.9102,C 0.0889,E1 0.9989,E2 504.1418} C_DIS
LIN {X 1.7934,Y -4.4645,Z 51,A -63.7551,B 0.9091,C 0.0995,E1 0.9807,E2 511.1775} C_DIS
LIN {X 1.1594,Y -4.6719,Z 51,A -71.2295,B 0.9081,C 0.1084,E1 0.9604,E2 518.6539} C_DIS
LIN {X 0.5024,Y -4.7874,Z 51,A -78.5821,B 0.9073,C 0.1147,E1 0.9398,E2 526.0077} C_DIS
LIN {X 0.5024,Y -4.7874,Z 51,A -78.5821,B 0.9073,C 0.1147,E1 0.9398,E2 526.0077} C_DIS
Enddeposition()
LIN {X 0.0023,Y -5.7178,Z 51,A -90.8411,B 8.9594,C -0.481,E1 8.9797,E2 536.7246} C_DIS
Startdeposition()
$VEL.CP = VEL_PRINT
LIN {X 1.0021,Y -5.6269,Z 51,A -80.9059,B 8.9592,C -0.4857,E1 9.0072,E2 526.7847} C_DIS
LIN {X 1.7805,Y -5.4292,Z 51,A -72.9864,B 8.9588,C -0.4928,E1 9.0285,E2 518.861} C_DIS
LIN {X 2.5242,Y -5.1262,Z 51,A -64.99,B 8.9582,C -0.5029,E1 9.0488,E2 510.8597} C_DIS
LIN {X 3.2179,Y -4.7216,Z 51,A -56.9781,B 8.9575,C -0.5158,E1 9.0678,E2 502.8425} C_DIS
LIN {X 3.8477,Y -4.2233,Z 51,A -49.1326,B 8.9566,C -0.5308,E1 9.0845,E2 494.9923} C_DIS
LIN {X 4.4037,Y -3.6436,Z 51,A -41.2824,B 8.9556,C -0.5478,E1 9.099,E2 487.1374} C_DIS
LIN {X 4.8716,Y -2.9906,Z 51,A -33.1277,B 8.9544,C -0.5676,E1 9.1116,E2 478.9765} C_DIS
LIN {X 5.2424,Y -2.2778,Z 51,A -25.144,B 8.9531,C -0.5883,E1 9.1212,E2 470.9876} C_DIS
LIN {X 5.5104,Y -1.5204,Z 51,A -17.3784,B 8.9517,C -0.6093,E1 9.1277,E2 463.2181} C_DIS
LIN {X 5.6694,Y -0.733,Z 51,A -9.4561,B 8.9502,C -0.6315,E1 9.1313,E2 455.2915} C_DIS
LIN {X 5.7158,Y 0.0692,Z 51,A -1.3739,B 8.9485,C -0.6544,E1 9.1318,E2 447.2047} C_DIS
LIN {X 5.6492,Y 0.8698,Z 51,A 6.3865,B 8.9469,C -0.676,E1 9.1292,E2 439.4417} C_DIS
LIN {X 5.4719,Y 1.6533,Z 51,A 14.3296,B 8.9453,C -0.6976,E1 9.1236,E2 431.4959} C_DIS
LIN {X 5.1852,Y 2.4037,Z 51,A 22.2873,B 8.9437,C -0.7181,E1 9.115,E2 423.536} C_DIS
LIN {X 4.7976,Y 3.1074,Z 51,A 30.2134,B 8.9421,C -0.7371,E1 9.1036,E2 415.6086} C_DIS
LIN {X 4.3144,Y 3.7493,Z 51,A 38.1666,B 8.9407,C -0.7543,E1 9.0896,E2 407.6548} C_DIS
LIN {X 3.7454,Y 4.3164,Z 51,A 46.1597,B 8.9394,C -0.7695,E1 9.0733,E2 399.6617} C_DIS
LIN {X 3.1027,Y 4.798,Z 51,A 54.1848,B 8.9383,C -0.7822,E1 9.0549,E2 391.6373} C_DIS
LIN {X 2.3994,Y 5.1859,Z 51,A 62.0998,B 8.9375,C -0.792,E1 9.0352,E2 383.7241} C_DIS
LIN {X 1.6488,Y 5.4718,Z 51,A 70.1541,B 8.9369,C -0.7991,E1 9.0139,E2 375.672} C_DIS
LIN {X 0.8651,Y 5.6476,Z 51,A 78.1447,B 8.9365,C -0.8031,E1 8.992,E2 367.6845} C_DIS
LIN {X 0.0648,Y 5.7136,Z 51,A 86.139,B 8.9365,C -0.8039,E1 8.9697,E2 359.6939} C_DIS
LIN {X -0.737,Y 5.6674,Z 51,A 94.2804,B 8.9366,C -0.8017,E1 8.9471,E2 351.5563} C_DIS
LIN {X -1.7188,Y 5.4563,Z 51,A 104.8879,B 8.9373,C -0.7941,E1 8.9185,E2 340.9528} C_DIS
LIN {X -2.7041,Y 5.0379,Z 51,A 112.8805,B 8.9383,C -0.783,E1 8.8982,E2 332.9769} C_DIS
LIN {X -3.3013,Y 4.672,Z 51,A 122.0974,B 8.9394,C -0.7701,E1 8.8765,E2 323.7571} C_DIS
LIN {X -3.764,Y 4.3033,Z 51,A 128.4283,B 8.9403,C -0.7587,E1 8.863,E2 317.4287} C_DIS
LIN {X -4.3194,Y 3.7437,Z 51,A 136.3621,B 8.9417,C -0.7421,E1 8.848,E2 309.5004} C_DIS
LIN {X -4.7937,Y 3.114,Z 51,A 144.3695,B 8.9433,C -0.7233,E1 8.8352,E2 301.4983} C_DIS
LIN {X -5.176,Y 2.4246,Z 51,A 152.1426,B 8.9448,C -0.7035,E1 8.8253,E2 293.731} C_DIS
LIN {X -5.4042,Y 1.8786,Z 51,A 159.0392,B 8.9462,C -0.6856,E1 8.8187,E2 286.835} C_DIS
LIN {X -5.6506,Y 0.8595,Z 51,A 168.8286,B 8.9483,C -0.6579,E1 8.8132,E2 277.0547} C_DIS
LIN {X -5.7142,Y 0.1403,Z 51,A 176.3089,B 8.9498,C -0.6369,E1 8.812,E2 269.5776} C_DIS
LIN {X -5.6707,Y -0.7614,Z 51,A -173.6357,B 8.9517,C -0.6093,E1 8.8146,E2 259.5231} C_DIS
LIN {X -5.4879,Y -1.6177,Z 51,A -164.3374,B 8.9533,C -0.5844,E1 8.8213,E2 250.2262} C_DIS
LIN {X -4.9438,Y -2.8815,Z 51,A -149.0601,B 8.9556,C -0.5475,E1 8.8406,E2 234.9465} C_DIS
LIN {X -4.1317,Y -3.9563,Z 51,A -137.1406,B 8.9572,C -0.5215,E1 8.8621,E2 223.0355} C_DIS
LIN {X -3.3223,Y -4.6575,Z 51,A -126.4818,B 8.9582,C -0.5035,E1 8.8853,E2 212.3768} C_DIS
LIN {X -2.561,Y -5.1095,Z 51,A -118.0929,B 8.9588,C -0.4925,E1 8.9058,E2 203.9887} C_DIS
LIN {X -1.9097,Y -5.3882,Z 51,A -110.8934,B 8.9592,C -0.4859,E1 8.9245,E2 196.7871} C_DIS
LIN {X -1.2286,Y -5.583,Z 51,A -103.5538,B 8.9594,C -0.4819,E1 8.9444,E2 189.4441} C_DIS
LIN {X -0.5284,Y -5.691,Z 51,A -96.6057,B 8.9594,C -0.4802,E1 8.9636,E2 182.4939} C_DIS
LIN {X -0.5284,Y -5.691,Z 51,A -96.6057,B 8.9594,C -0.4802,E1 8.9636,E2 182.4939} C_DIS
Enddeposition()
LIN {X 0.0089,Y -6.6205,Z 51,A -96.6921,B 17.1883,C -1.5891,E1 17.2563,E2 180.7949} C_DIS
Startdeposition()
$VEL.CP = VEL_PRINT
LIN {X -0.8772,Y -6.5613,Z 51,A -104.4299,B 17.1883,C -1.5898,E1 17.2348,E2 188.5359} C_DIS
LIN {X -1.5752,Y -6.4283,Z 51,A -110.7976,B 17.188,C -1.5924,E1 17.2174,E2 194.9063} C_DIS
LIN {X -2.2552,Y -6.222,Z 51,A -116.8503,B 17.1876,C -1.5972,E1 17.2014,E2 200.9594} C_DIS
LIN {X -2.9102,Y -5.9461,Z 51,A -122.767,B 17.187,C -1.6038,E1 17.1863,E2 206.8753} C_DIS
LIN {X -3.5314,Y -5.6011,Z 51,A -129.3176,B 17.1863,C -1.6121,E1 17.1706,E2 213.4274} C_DIS
LIN {X -4.1108,Y -5.1896,Z 51,A -135.3562,B 17.1854,C -1.6221,E1 17.1571,E2 219.4642} C_DIS
LIN {X -4.6431,Y -4.7188,Z 51,A -141.7361,B 17.1843,C -1.6339,E1 17.1441,E2 225.8433} C_DIS
LIN {X -5.1216,Y -4.1932,Z 51,A -147.7651,B 17.1831,C -1.6469,E1 17.1331,E2 231.8691} C_DIS
LIN {X -5.5417,Y -3.62,Z 51,A -153.9303,B 17.1817,C -1.6612,E1 17.1233,E2 238.0312} C_DIS
LIN {X -5.8984,Y -3.0053,Z 51,A -160.3777,B 17.1802,C -1.6769,E1 17.1147,E2 244.4761} C_DIS
LIN {X -6.1845,Y -2.3549,Z 51,A -166.3891,B 17.1787,C -1.6931,E1 17.1083,E2 250.4824} C_DIS
LIN {X -6.4037,Y -1.6788,Z 51,A -172.6009,B 17.1771,C -1.7103,E1 17.1035,E2 256.6896} C_DIS
LIN {X -6.5447,Y -0.9823,Z 51,A -178.6162,B 17.1754,C -1.7277,E1 17.1005,E2 262.699} C_DIS
LIN {X -6.6153,Y -0.2753,Z 51,A 175.0242,B 17.1736,C -1.746,E1 17.0992,E2 269.0538} C_DIS
LIN {X -6.6073,Y 0.4353,Z 51,A 168.6995,B 17.1718,C -1.7643,E1 17.0999,E2 275.3731} C_DIS
LIN {X -6.5221,Y 1.1409,Z 51,A 162.4669,B 17.1699,C -1.7824,E1 17.1025,E2 281.5997} C_DIS
LIN {X -6.3618,Y 1.8333,Z 51,A 156.3221,B 17.1682,C -1.8001,E1 17.1068,E2 287.738} C_DIS
LIN {X -6.1289,Y 2.5046,Z 51,A 150.0754,B 17.1664,C -1.8174,E1 17.1129,E2 293.9785} C_DIS
LIN {X -5.8245,Y 3.1468,Z 51,A 143.7031,B 17.1647,C -1.8341,E1 17.121,E2 300.345} C_DIS
LIN {X -5.4517,Y 3.7519,Z 51,A 137.7458,B 17.1631,C -1.8495,E1 17.13,E2 306.2949} C_DIS
LIN {X -5.0183,Y 4.315,Z 51,A 131.4846,B 17.1615,C -1.8641,E1 17.141,E2 312.55} C_DIS
LIN {X -4.5272,Y 4.8286,Z 51,A 125.3765,B 17.1601,C -1.8773,E1 17.1531,E2 318.6517} C_DIS
LIN {X -3.9844,Y 5.2872,Z 51,A 119.0605,B 17.1589,C -1.8892,E1 17.1669,E2 324.9624} C_DIS
LIN {X -3.3945,Y 5.6836,Z 51,A 112.8843,B 17.1578,C -1.8995,E1 17.1814,E2 331.133} C_DIS
LIN {X -2.7658,Y 6.0146,Z 51,A 106.7596,B 17.1568,C -1.9082,E1 17.1967,E2 337.2524} C_DIS
LIN {X -2.105,Y 6.2763,Z 51,A 100.5683,B 17.1561,C -1.915,E1 17.2129,E2 343.439} C_DIS
LIN {X -1.4204,Y 6.4672,Z 51,A 94.4185,B 17.1555,C -1.9201,E1 17.2296,E2 349.5846} C_DIS
LIN {X -0.7191,Y 6.5821,Z 51,A 88.1054,B 17.1552,C -1.9231,E1 17.247,E2 355.8946} C_DIS
LIN {X -0.0093,Y 6.6197,Z 51,A 81.8247,B 17.1551,C -1.9241,E1 17.2646,E2 362.1727} C_DIS
LIN {X 0.7002,Y 6.581,Z 51,A 76.0403,B 17.1551,C -1.924,E1 17.2806,E2 367.953} C_DIS
LIN {X 1.4018,Y 6.469,Z 51,A 69.7875,B 17.1554,C -1.9212,E1 17.2978,E2 374.2045} C_DIS
LIN {X 2.0875,Y 6.282,Z 51,A 63.4691,B 17.1559,C -1.9163,E1 17.3147,E2 380.5226} C_DIS
LIN {X 2.7488,Y 6.0216,Z 51,A 57.5634,B 17.1566,C -1.9105,E1 17.3298,E2 386.4267} C_DIS
LIN {X 3.3788,Y 5.6926,Z 51,A 51.4243,B 17.1574,C -1.9024,E1 17.3448,E2 392.5661} C_DIS
LIN {X 3.9696,Y 5.2977,Z 51,A 45.2241,B 17.1585,C -1.8924,E1 17.359,E2 398.7676} C_DIS
LIN {X 4.5144,Y 4.8412,Z 51,A 39.1884,B 17.1597,C -1.8814,E1 17.3716,E2 404.8044} C_DIS
LIN {X 5.0079,Y 4.3299,Z 51,A 32.7157,B 17.1612,C -1.8675,E1 17.3838,E2 411.2812} C_DIS
LIN {X 5.4433,Y 3.768,Z 51,A 27.2327,B 17.1624,C -1.8559,E1 17.3928,E2 416.7637} C_DIS
LIN {X 5.8165,Y 3.1633,Z 51,A 20.4623,B 17.1642,C -1.8382,E1 17.4023,E2 423.5411} C_DIS
LIN {X 6.1196,Y 2.5205,Z 51,A 14.9089,B 17.1657,C -1.8245,E1 17.4086,E2 429.0954} C_DIS
LIN {X 6.3565,Y 1.8504,Z 51,A 8.4362,B 17.1675,C -1.8061,E1 17.4141,E2 435.5748} C_DIS
LIN {X 6.5161,Y 1.1579,Z 51,A 2.4684,B 17.1692,C -1.7894,E1 17.4175,E2 441.5467} C_DIS
LIN {X 6.6047,Y 0.4528,Z 51,A -3.5493,B 17.171,C -1.772,E1 17.4191,E2 447.5693} C_DIS
LIN {X 6.6139,Y -0.2578,Z 51,A -9.5606,B 17.1727,C -1.7546,E1 17.4189,E2 453.5858} C_DIS
LIN {X 6.5502,Y -0.9655,Z 51,A -15.7572,B 17.1745,C -1.7363,E1 17.4169,E2 459.7891} C_DIS
LIN {X 6.4088,Y -1.662,Z 51,A -21.9787,B 17.1763,C -1.7181,E1 17.413,E2 466.0174} C_DIS
LIN {X 6.1931,Y -2.3392,Z 51,A -27.9451,B 17.1779,C -1.7015,E1 17.4075,E2 471.9893} C_DIS
LIN {X 5.9066,Y -2.9895,Z 51,A -34.0899,B 17.1795,C -1.6848,E1 17.4001,E2 478.1407} C_DIS
LIN {X 5.552,Y -3.6053,Z 51,A -40.175,B 17.181,C -1.6691,E1 17.3913,E2 484.2321} C_DIS
LIN {X 5.1338,Y -4.1798,Z 51,A -46.2438,B 17.1824,C -1.6545,E1 17.3809,E2 490.307} C_DIS
LIN {X 4.6562,Y -4.706,Z 51,A -52.4497,B 17.1837,C -1.6405,E1 17.3689,E2 496.5196} C_DIS
LIN {X 4.1247,Y -5.1779,Z 51,A -58.4598,B 17.1848,C -1.6286,E1 17.3561,E2 502.535} C_DIS
LIN {X 3.5459,Y -5.5904,Z 51,A -64.7904,B 17.1858,C -1.6171,E1 17.3414,E2 508.8725} C_DIS
LIN {X 2.9251,Y -5.9361,Z 51,A -70.7247,B 17.1866,C -1.6085,E1 17.3267,E2 514.8108} C_DIS
LIN {X 2.2721,Y -6.2162,Z 51,A -76.7228,B 17.1873,C -1.6012,E1 17.3112,E2 520.813} C_DIS
LIN {X 1.5927,Y -6.4249,Z 51,A -83.0874,B 17.1878,C -1.5949,E1 17.294,E2 527.1834} C_DIS
LIN {X 0.8947,Y -6.5587,Z 51,A -88.8978,B 17.1881,C -1.5916,E1 17.278,E2 532.9958} C_DIS
LIN {X 0.0089,Y -6.6205,Z 51,A -94.2864,B 17.188,C -1.593,E1 17.263,E2 538.376} C_DIS
Enddeposition()
LIN {X 0.0089,Y -6.6205,Z 51,A -94.2864,B 17.188,C -1.593,E1 17.263,E2 538.376} C_DIS
Startdeposition()
$VEL.CP = VEL_PRINT
LIN {X 0.6295,Y -7.5004,Z 51,A -90.603,B 24.8118,C -3.1636,E1 25.0195,E2 532.7398} C_DIS
LIN {X 1.5633,Y -7.3614,Z 51,A -83.7314,B 24.8113,C -3.1682,E1 25.0384,E2 525.8649} C_DIS
LIN {X 2.653,Y -7.0389,Z 51,A -75.1261,B 24.81,C -3.1782,E1 25.0612,E2 517.252} C_DIS
LIN {X 3.4004,Y -6.708,Z 51,A -69.1447,B 24.809,C -3.1868,E1 25.0763,E2 511.2657} C_DIS
LIN {X 4.1084,Y -6.2996,Z 51,A -63.0175,B 24.8077,C -3.1977,E1 25.0909,E2 505.132} C_DIS
LIN {X 4.7685,Y -5.8177,Z 51,A -56.7028,B 24.8061,C -3.211,E1 25.1049,E2 498.8089} C_DIS
LIN {X 5.5153,Y -5.1203,Z 51,A -48.6898,B 24.8037,C -3.2303,E1 25.1207,E2 490.7839} C_DIS
LIN {X 6.3335,Y -4.0661,Z 51,A -37.9554,B 24.8001,C -3.2601,E1 25.1382,E2 480.0309} C_DIS
LIN {X 6.9472,Y -2.8859,Z 51,A -30.2791,B 24.7981,C -3.2761,E1 25.1477,E2 472.3577} C_DIS
LIN {X 7.1999,Y -2.1903,Z 51,A -22.7444,B 24.7947,C -3.3034,E1 25.1544,E2 464.8007} C_DIS
LIN {X 7.4262,Y -1.1864,Z 51,A -15.4966,B 24.7921,C -3.3243,E1 25.1584,E2 457.5456} C_DIS
LIN {X 7.5127,Y -0.3677,Z 51,A -9.3058,B 24.7897,C -3.3433,E1 25.1597,E2 451.3464} C_DIS
LIN {X 7.4883,Y 0.7553,Z 51,A -0.4231,B 24.7861,C -3.3714,E1 25.1584,E2 442.4499} C_DIS
LIN {X 7.3331,Y 1.6984,Z 51,A 7.1448,B 24.7831,C -3.3947,E1 25.1542,E2 434.8706} C_DIS
LIN {X 6.9877,Y 2.7849,Z 51,A 15.1794,B 24.7804,C -3.4161,E1 25.1468,E2 426.8305} C_DIS
LIN {X 6.6405,Y 3.5342,Z 51,A 21.3757,B 24.7783,C -3.4325,E1 25.1391,E2 420.6284} C_DIS
LIN {X 6.0164,Y 4.521,Z 51,A 30.4377,B 24.7753,C -3.455,E1 25.1249,E2 411.5576} C_DIS
LIN {X 5.3273,Y 5.3103,Z 51,A 38.2921,B 24.7731,C -3.4716,E1 25.1101,E2 403.6984} C_DIS
LIN {X 4.7031,Y 5.8699,Z 51,A 44.5309,B 24.7717,C -3.4828,E1 25.0968,E2 397.4572} C_DIS
LIN {X 3.7376,Y 6.5328,Z 51,A 53.8817,B 24.7697,C -3.4978,E1 25.0748,E2 388.101} C_DIS
LIN {X 2.6786,Y 7.0292,Z 51,A 60.6185,B 24.7694,C -3.5,E1 25.0577,E2 381.3759} C_DIS
LIN {X 1.9393,Y 7.2715,Z 51,A 68.3513,B 24.7681,C -3.5099,E1 25.037,E2 373.6333} C_DIS
LIN {X 1.119,Y 7.4424,Z 51,A 75.1981,B 24.7676,C -3.5134,E1 25.0182,E2 366.7854} C_DIS
LIN {X 0.113,Y 7.5252,Z 51,A 82.8638,B 24.7676,C -3.513,E1 24.9968,E2 359.1232} C_DIS
LIN {X -0.9896,Y 7.4617,Z 51,A 90.9454,B 24.7683,C -3.5083,E1 24.9744,E2 351.0486} C_DIS
LIN {X -1.9987,Y 7.2508,Z 51,A 98.6286,B 24.7692,C -3.5012,E1 24.9535,E2 343.3723} C_DIS
LIN {X -2.973,Y 6.9133,Z 51,A 107.0841,B 24.7705,C -3.4916,E1 24.9316,E2 334.9215} C_DIS
LIN {X -4.0241,Y 6.3595,Z 51,A 115.948,B 24.7726,C -3.4761,E1 24.9101,E2 326.0687} C_DIS
LIN {X -4.8357,Y 5.7587,Z 51,A 123.2202,B 24.7746,C -3.4603,E1 24.8941,E2 318.8078} C_DIS
LIN {X -5.4269,Y 5.2081,Z 51,A 129.3147,B 24.7765,C -3.446,E1 24.882,E2 312.7218} C_DIS
LIN {X -6.1454,Y 4.344,Z 51,A 137.2281,B 24.7793,C -3.4243,E1 24.8683,E2 304.8234} C_DIS
LIN {X -6.641,Y 3.5393,Z 51,A 145.22,B 24.7819,C -3.4042,E1 24.8569,E2 296.8384} C_DIS
LIN {X -7.0381,Y 2.6651,Z 51,A 153.3615,B 24.7847,C -3.3824,E1 24.8482,E2 288.704} C_DIS
LIN {X -7.3239,Y 1.7327,Z 51,A 160.7048,B 24.7876,C -3.3599,E1 24.8429,E2 281.372} C_DIS
LIN {X -7.4962,Y 0.5959,Z 51,A 169.1457,B 24.791,C -3.3331,E1 24.84,E2 272.9449} C_DIS
LIN {X -7.5161,Y -0.2549,Z 51,A 175.6338,B 24.7935,C -3.3131,E1 24.84,E2 266.4658} C_DIS
LIN {X -7.411,Y -1.3137,Z 51,A -175.5301,B 24.7966,C -3.288,E1 24.8435,E2 257.6372} C_DIS
LIN {X -7.1209,Y -2.4247,Z 51,A -167.4496,B 24.7997,C -3.2629,E1 24.8498,E2 249.5702} C_DIS
LIN {X -6.8271,Y -3.1577,Z 51,A -161.2923,B 24.8018,C -3.2463,E1 24.8566,E2 243.4186} C_DIS
LIN {X -6.4587,Y -3.8562,Z 51,A -155.3093,B 24.8037,C -3.2307,E1 24.8648,E2 237.4416} C_DIS
LIN {X -6.0182,Y -4.5114,Z 51,A -149.3784,B 24.8054,C -3.2163,E1 24.8743,E2 231.5162} C_DIS
LIN {X -5.5127,Y -5.118,Z 51,A -143.0842,B 24.807,C -3.2033,E1 24.886,E2 225.2249} C_DIS
LIN {X -4.9456,Y -5.6675,Z 51,A -137.3511,B 24.8084,C -3.1915,E1 24.8977,E2 219.4968} C_DIS
LIN {X -4.3244,Y -6.1548,Z 51,A -131.0852,B 24.8096,C -3.1817,E1 24.9118,E2 213.232} C_DIS
LIN {X -3.4838,Y -6.6723,Z 51,A -122.9173,B 24.8107,C -3.1724,E1 24.9316,E2 205.0626} C_DIS
LIN {X -2.3708,Y -7.1381,Z 51,A -114.1998,B 24.8118,C -3.1634,E1 24.9543,E2 196.348} C_DIS
LIN {X -1.5025,Y -7.3709,Z 51,A -107.3095,B 24.8122,C -3.1602,E1 24.973,E2 189.4563} C_DIS
LIN {X -0.8366,Y -7.4791,Z 51,A -102.1531,B 24.8123,C -3.1593,E1 24.9873,E2 184.2982} C_DIS
LIN {X -0.0001,Y -7.5234,Z 51,A -98.0536,B 24.8129,C -3.1541,E1 24.9987,E2 180.2102} C_DIS
Enddeposition()
LIN {X -0.0001,Y -7.5234,Z 51,A -98.0536,B 24.8129,C -3.1541,E1 24.9987,E2 180.2102} C_DIS
Startdeposition()
$VEL.CP = VEL_PRINT
LIN {X -0.6694,Y -8.3984,Z 51,A -103.6165,B 24.8152,C -3.1354,E1 24.9831,E2 185.8195} C_DIS
LIN {X -1.5204,Y -8.2855,Z 51,A -109.2737,B 24.8149,C -3.1374,E1 24.9675,E2 191.477} C_DIS
LIN {X -2.3558,Y -8.0881,Z 51,A -115.1071,B 24.8145,C -3.1407,E1 24.9517,E2 197.3112} C_DIS
LIN {X -3.1668,Y -7.8071,Z 51,A -120.957,B 24.8139,C -3.1458,E1 24.9364,E2 203.161} C_DIS
LIN {X -3.9449,Y -7.4443,Z 51,A -126.8454,B 24.8131,C -3.1526,E1 24.9217,E2 209.0488} C_DIS
LIN {X -4.6819,Y -7.0042,Z 51,A -132.7191,B 24.8121,C -3.1611,E1 24.9079,E2 214.9208} C_DIS
LIN {X -5.3701,Y -6.4912,Z 51,A -138.5786,B 24.8109,C -3.1712,E1 24.895,E2 220.7777} C_DIS
LIN {X -6.2066,Y -5.7029,Z 51,A -146.7183,B 24.809,C -3.1868,E1 24.879,E2 228.9145} C_DIS
LIN {X -6.8737,Y -4.8697,Z 51,A -153.8181,B 24.807,C -3.2039,E1 24.867,E2 236.0072} C_DIS
LIN {X -7.3322,Y -4.1492,Z 51,A -159.4691,B 24.8052,C -3.2186,E1 24.8589,E2 241.652} C_DIS
LIN {X -7.7154,Y -3.386,Z 51,A -165.3924,B 24.8032,C -3.2343,E1 24.8518,E2 247.5698} C_DIS
LIN {X -8.1312,Y -2.219,Z 51,A -174.2022,B 24.8003,C -3.2586,E1 24.8443,E2 256.3719} C_DIS
LIN {X -8.3433,Y -1.2008,Z 51,A 178.4965,B 24.7976,C -3.28,E1 24.8407,E2 263.6653} C_DIS
LIN {X -8.4266,Y -0.167,Z 51,A 171.7024,B 24.7949,C -3.3016,E1 24.8398,E2 270.4484} C_DIS
LIN {X -8.3797,Y 0.9038,Z 51,A 164.3228,B 24.7921,C -3.3242,E1 24.8413,E2 277.8181} C_DIS
LIN {X -8.2501,Y 1.7228,Z 51,A 157.7829,B 24.7899,C -3.342,E1 24.8447,E2 284.354} C_DIS
LIN {X -7.8897,Y 2.964,Z 51,A 149.7985,B 24.7866,C -3.368,E1 24.8517,E2 292.3217} C_DIS
LIN {X -7.3357,Y 4.1503,Z 51,A 140.8775,B 24.7833,C -3.3934,E1 24.8628,E2 301.2298} C_DIS
LIN {X -6.7184,Y 5.0853,Z 51,A 133.2598,B 24.7807,C -3.4136,E1 24.875,E2 308.8364} C_DIS
LIN {X -6.0473,Y 5.8706,Z 51,A 126.0538,B 24.7785,C -3.4305,E1 24.8884,E2 316.0339} C_DIS
LIN {X -5.2294,Y 6.61,Z 51,A 118.9127,B 24.7764,C -3.4469,E1 24.9035,E2 323.1636} C_DIS
LIN {X -4.6452,Y 7.0341,Z 51,A 113.4079,B 24.7752,C -3.4558,E1 24.9162,E2 328.6656} C_DIS
LIN {X -3.6475,Y 7.5977,Z 51,A 105.7471,B 24.7736,C -3.4685,E1 24.9351,E2 336.3172} C_DIS
LIN {X -2.6175,Y 8.0118,Z 51,A 98.0356,B 24.7723,C -3.4777,E1 24.9553,E2 344.0224} C_DIS
LIN {X -1.4588,Y 8.2979,Z 51,A 90.2726,B 24.7713,C -3.4853,E1 24.9764,E2 351.777} C_DIS
LIN {X -0.2034,Y 8.4258,Z 51,A 81.6952,B 24.7709,C -3.4889,E1 25.0003,E2 360.3493} C_DIS
LIN {X 0.8115,Y 8.3847,Z 51,A 74.9594,B 24.7708,C -3.4895,E1 25.019,E2 367.0811} C_DIS
LIN {X 1.6159,Y 8.2693,Z 51,A 69.3165,B 24.7711,C -3.4873,E1 25.0346,E2 372.7233} C_DIS
LIN {X 2.6911,Y 7.9887,Z 51,A 61.0374,B 24.7721,C -3.4796,E1 25.0567,E2 381.0064} C_DIS
LIN {X 3.8563,Y 7.4898,Z 51,A 52.9288,B 24.7731,C -3.4719,E1 25.0773,E2 389.1127} C_DIS
LIN {X 4.8561,Y 6.8885,Z 51,A 44.9498,B 24.7747,C -3.4597,E1 25.096,E2 397.0948} C_DIS
LIN {X 5.7465,Y 6.1629,Z 51,A 37.3175,B 24.7765,C -3.446,E1 25.1121,E2 404.73} C_DIS
LIN {X 6.3152,Y 5.5758,Z 51,A 31.9293,B 24.7779,C -3.4349,E1 25.1224,E2 410.1207} C_DIS
LIN {X 7.0095,Y 4.681,Z 51,A 23.6574,B 24.7807,C -3.4136,E1 25.1359,E2 418.4032} C_DIS
LIN {X 7.5605,Y 3.7242,Z 51,A 16.6146,B 24.7829,C -3.3963,E1 25.1452,E2 425.4501} C_DIS
LIN {X 7.9129,Y 2.901,Z 51,A 10.4653,B 24.7852,C -3.3789,E1 25.1516,E2 431.6066} C_DIS
LIN {X 8.2246,Y 1.8275,Z 51,A 4.8193,B 24.7866,C -3.3677,E1 25.1558,E2 437.2468} C_DIS
LIN {X 8.3634,Y 1.0475,Z 51,A -2.4927,B 24.7901,C -3.3404,E1 25.1591,E2 444.5808} C_DIS
LIN {X 8.4299,Y -0.0108,Z 51,A -10.0014,B 24.7931,C -3.3163,E1 25.1597,E2 452.1018} C_DIS
LIN {X 8.345,Y -1.186,Z 51,A -18.2025,B 24.7963,C -3.2904,E1 25.1572,E2 460.3158} C_DIS
LIN {X 8.0971,Y -2.3446,Z 51,A -25.1048,B 24.7986,C -3.2724,E1 25.1526,E2 467.2212} C_DIS
LIN {X 7.8489,Y -3.0747,Z 51,A -30.8072,B 24.8008,C -3.2541,E1 25.1471,E2 472.9349} C_DIS
LIN {X 7.2867,Y -4.2375,Z 51,A -40.2337,B 24.8043,C -3.2256,E1 25.1348,E2 482.3793} C_DIS
LIN {X 6.6619,Y -5.162,Z 51,A -47.0557,B 24.8062,C -3.2097,E1 25.1236,E2 489.2062} C_DIS
LIN {X 5.8896,Y -6.0237,Z 51,A -54.7612,B 24.8084,C -3.1916,E1 25.1088,E2 496.9209} C_DIS
LIN {X 5.2415,Y -6.5943,Z 51,A -60.473,B 24.8099,C -3.1797,E1 25.0966,E2 502.639} C_DIS
LIN {X 4.5395,Y -7.0971,Z 51,A -66.3409,B 24.8112,C -3.1684,E1 25.083,E2 508.514} C_DIS
LIN {X 3.5966,Y -7.6224,Z 51,A -73.9252,B 24.8128,C -3.1554,E1 25.0642,E2 516.1082} C_DIS
LIN {X 2.5614,Y -8.0294,Z 51,A -81.3425,B 24.8139,C -3.1464,E1 25.0447,E2 523.5316} C_DIS
LIN {X 1.6141,Y -8.2729,Z 51,A -87.8701,B 24.8145,C -3.1408,E1 25.0269,E2 530.0637} C_DIS
LIN {X 0.597,Y -8.4071,Z 51,A -95.2086,B 24.8151,C -3.1358,E1 25.0065,E2 537.4092} C_DIS
LIN {X 0.597,Y -8.4071,Z 51,A -95.2086,B 24.8151,C -3.1358,E1 25.0065,E2 537.4092} C_DIS
Enddeposition()
LIN {X -0.0418,Y -9.3301,Z 51,A -96.452,B 24.816,C -3.1285,E1 25.003,E2 538.6696} C_DIS
Startdeposition()
$VEL.CP = VEL_PRINT
LIN {X 0.951,Y -9.2826,Z 51,A -89.8376,B 24.8154,C -3.1331,E1 25.0214,E2 532.0474} C_DIS
LIN {X 2.1527,Y -9.076,Z 51,A -84.0803,B 24.8155,C -3.1324,E1 25.0372,E2 526.2985} C_DIS
LIN {X 2.8947,Y -8.8707,Z 51,A -77.9839,B 24.8142,C -3.1432,E1 25.0536,E2 520.1868} C_DIS
LIN {X 4.14,Y -8.3617,Z 51,A -69.5557,B 24.8127,C -3.156,E1 25.0751,E2 511.7487} C_DIS
LIN {X 5.1927,Y -7.7491,Z 51,A -62.2719,B 24.8112,C -3.1686,E1 25.0925,E2 504.4579} C_DIS
LIN {X 6.1602,Y -7.0084,Z 51,A -54.8107,B 24.8093,C -3.1844,E1 25.1087,E2 496.9875} C_DIS
LIN {X 6.9531,Y -6.2175,Z 51,A -48.0089,B 24.8074,C -3.2005,E1 25.1218,E2 490.1769} C_DIS
LIN {X 7.7066,Y -5.2596,Z 51,A -40.4722,B 24.805,C -3.2203,E1 25.1344,E2 482.6293} C_DIS
LIN {X 8.4027,Y -4.0556,Z 51,A -31.8452,B 24.8019,C -3.245,E1 25.1459,E2 473.9889} C_DIS
LIN {X 8.862,Y -2.9113,Z 51,A -24.5373,B 24.7994,C -3.2659,E1 25.153,E2 466.6721} C_DIS
LIN {X 9.1723,Y -1.7204,Z 51,A -16.9533,B 24.7965,C -3.2892,E1 25.1578,E2 459.0769} C_DIS
LIN {X 9.3051,Y -0.6923,Z 51,A -10.7835,B 24.7942,C -3.3078,E1 25.1596,E2 452.8995} C_DIS
LIN {X 9.3201,Y 0.3727,Z 51,A -4.3159,B 24.7917,C -3.3276,E1 25.1595,E2 446.4234} C_DIS
LIN {X 9.2199,Y 1.4332,Z 51,A 2.5989,B 24.7889,C -3.3498,E1 25.1571,E2 439.4968} C_DIS
LIN {X 8.9482,Y 2.6343,Z 51,A 9.7965,B 24.7863,C -3.37,E1 25.1521,E2 432.2929} C_DIS
LIN {X 8.5318,Y 3.7791,Z 51,A 17.2634,B 24.7836,C -3.3908,E1 25.1445,E2 424.8179} C_DIS
LIN {X 7.8985,Y 4.9671,Z 51,A 25.6647,B 24.7808,C -3.413,E1 25.1329,E2 416.4075} C_DIS
LIN {X 7.1813,Y 5.9531,Z 51,A 32.9359,B 24.7787,C -3.4293,E1 25.1206,E2 409.1319} C_DIS
LIN {X 6.4168,Y 6.7732,Z 51,A 40.021,B 24.7767,C -3.4445,E1 25.1067,E2 402.0409} C_DIS
LIN {X 5.5768,Y 7.4815,Z 51,A 46.6306,B 24.7752,C -3.4558,E1 25.0922,E2 395.4292} C_DIS
LIN {X 4.9211,Y 7.9269,Z 51,A 51.6116,B 24.7742,C -3.4636,E1 25.0805,E2 390.4457} C_DIS
LIN {X 3.8446,Y 8.4984,Z 51,A 58.7954,B 24.7732,C -3.4714,E1 25.0626,E2 383.2627} C_DIS
LIN {X 2.7048,Y 8.9301,Z 51,A 66.2762,B 24.7724,C -3.4776,E1 25.0428,E2 375.7822} C_DIS
LIN {X 1.3917,Y 9.2266,Z 51,A 74.7314,B 24.7718,C -3.4817,E1 25.0197,E2 367.3275} C_DIS
LIN {X 0.1639,Y 9.3279,Z 51,A 82.1725,B 24.7718,C -3.4812,E1 24.999,E2 359.8904} C_DIS
LIN {X -0.9604,Y 9.2815,Z 51,A 89.3841,B 24.7722,C -3.4791,E1 24.9789,E2 352.681} C_DIS
LIN {X -1.9452,Y 9.1255,Z 51,A 95.3603,B 24.7728,C -3.4741,E1 24.9625,E2 346.7102} C_DIS
LIN {X -3.1112,Y 8.7941,Z 51,A 102.6632,B 24.7739,C -3.4657,E1 24.9431,E2 339.4148} C_DIS
LIN {X -4.1526,Y 8.3556,Z 51,A 109.7982,B 24.7752,C -3.4559,E1 24.925,E2 332.2858} C_DIS
LIN {X -5.2021,Y 7.743,Z 51,A 117.1493,B 24.777,C -3.4424,E1 24.9076,E2 324.9439} C_DIS
LIN {X -6.1662,Y 7.0033,Z 51,A 124.7493,B 24.779,C -3.4268,E1 24.8911,E2 317.3526} C_DIS
LIN {X -6.9806,Y 6.1857,Z 51,A 131.6555,B 24.7812,C -3.41,E1 24.8778,E2 310.457} C_DIS
LIN {X -7.6492,Y 5.3426,Z 51,A 138.6967,B 24.7834,C -3.393,E1 24.8661,E2 303.4226} C_DIS
LIN {X -8.2755,Y 4.3036,Z 51,A 144.5113,B 24.7861,C -3.372,E1 24.8579,E2 297.6283} C_DIS
LIN {X -8.6058,Y 3.6051,Z 51,A 150.6789,B 24.7878,C -3.3583,E1 24.8508,E2 291.4596} C_DIS
LIN {X -8.9673,Y 2.5846,Z 51,A 158.091,B 24.7903,C -3.3383,E1 24.8445,E2 284.0529} C_DIS
LIN {X -9.22,Y 1.4327,Z 51,A 164.8389,B 24.7931,C -3.3161,E1 24.8411,E2 277.3184} C_DIS
LIN {X -9.3217,Y 0.4434,Z 51,A 171.2349,B 24.7955,C -3.2971,E1 24.8398,E2 270.9294} C_DIS
LIN {X -9.2958,Y -0.7758,Z 51,A 178.4035,B 24.7983,C -3.2741,E1 24.8407,E2 263.7728} C_DIS
LIN {X -9.1179,Y -1.9814,Z 51,A -174.0702,B 24.8011,C -3.2516,E1 24.8443,E2 256.2561} C_DIS
LIN {X -8.7382,Y -3.2713,Z 51,A -165.5416,B 24.804,C -3.2278,E1 24.8516,E2 247.7355} C_DIS
LIN {X -8.2357,Y -4.3804,Z 51,A -158.1883,B 24.8065,C -3.2077,E1 24.8606,E2 240.3907} C_DIS
LIN {X -7.5571,Y -5.4755,Z 51,A -149.9669,B 24.8088,C -3.1883,E1 24.8732,E2 232.1744} C_DIS
LIN {X -6.8727,Y -6.3058,Z 51,A -143.7013,B 24.8106,C -3.1736,E1 24.8846,E2 225.9158} C_DIS
LIN {X -6.0142,Y -7.1334,Z 51,A -136.2291,B 24.8123,C -3.1596,E1 24.9,E2 218.447} C_DIS
LIN {X -4.9271,Y -7.9232,Z 51,A -127.6677,B 24.8138,C -3.1471,E1 24.9197,E2 209.8866} C_DIS
LIN {X -3.9946,Y -8.4324,Z 51,A -121.3625,B 24.8148,C -3.1388,E1 24.9354,E2 203.5842} C_DIS
LIN {X -3.2159,Y -8.7586,Z 51,A -115.9711,B 24.8153,C -3.1345,E1 24.9494,E2 198.1914} C_DIS
LIN {X -2.2652,Y -9.0517,Z 51,A -109.9171,B 24.8157,C -3.1307,E1 24.9657,E2 192.1372} C_DIS
LIN {X -1.3848,Y -9.2277,Z 51,A -104.4161,B 24.8159,C -3.129,E1 24.9808,E2 186.6349} C_DIS
LIN {X -0.0418,Y -9.3301,Z 51,A -98.7401,B 24.8168,C -3.1211,E1 24.9966,E2 180.9754} C_DIS
Enddeposition()
LIN {X 0.0025,Y -4.8154,Z 52,A -2.8508,B 0,C 0,E1 0.1598,E2 90.0717} C_DIS
Startdeposition()
$VEL.CP = VEL_PRINT
LIN {X 0.8227,Y -4.7396,Z 52,A -2.8176,B 0,C 0,E1 0.1598,E2 90.0718} C_DIS
LIN {X 1.4625,Y -4.5823,Z 52,A -2.7874,B 0,C 0,E1 0.1598,E2 90.0718} C_DIS
LIN {X 2.0747,Y -4.3391,Z 52,A -2.7545,B 0,C 0,E1 0.1598,E2 90.0718} C_DIS
LIN {X 2.649,Y -4.0159,Z 52,A -2.7196,B 0,C 0,E1 0.1598,E2 90.0718} C_DIS
LIN {X 3.1732,Y -3.6168,Z 52,A -2.6833,B 0,C 0,E1 0.1598,E2 90.0719} C_DIS
LIN {X 3.6353,Y -3.1472,Z 52,A -2.6463,B 0,C 0,E1 0.1598,E2 90.0719} C_DIS
LIN {X 4.0326,Y -2.6216,Z 52,A -2.6092,B 0,C 0,E1 0.1598,E2 90.0719} C_DIS
LIN {X 4.3523,Y -2.0456,Z 52,A -2.5729,B 0,C 0,E1 0.1598,E2 90.0719} C_DIS
LIN {X 4.5925,Y -1.432,Z 52,A -2.5378,B 0,C 0,E1 0.1598,E2 90.0719} C_DIS
LIN {X 4.745,Y -0.791,Z 52,A -2.5048,B 0,C 0,E1 0.1598,E2 90.072} C_DIS
LIN {X 4.8093,Y -0.1352,Z 52,A -2.4745,B 0,C 0,E1 0.1598,E2 90.072} C_DIS
LIN {X 4.7835,Y 0.5233,Z 52,A -2.4473,B 0,C 0,E1 0.1598,E2 90.072} C_DIS
LIN {X 4.6667,Y 1.1719,Z 52,A -2.424,B 0,C 0,E1 0.1598,E2 90.072} C_DIS
LIN {X 4.462,Y 1.7983,Z 52,A -2.4048,B 0,C 0,E1 0.1598,E2 90.0721} C_DIS
LIN {X 4.1734,Y 2.3907,Z 52,A -2.3902,B 0,C 0,E1 0.1598,E2 90.0721} C_DIS
LIN {X 3.8079,Y 2.9389,Z 52,A -2.3803,B 0,C 0,E1 0.1598,E2 90.0722} C_DIS
LIN {X 3.3698,Y 3.4308,Z 52,A -2.3755,B 0,C 0,E1 0.1598,E2 90.0722} C_DIS
LIN {X 2.8704,Y 3.8606,Z 52,A -2.3756,B 0,C 0,E1 0.1598,E2 90.0722} C_DIS
LIN {X 2.3143,Y 4.2141,Z 52,A -2.3811,B 0,C 0,E1 0.1598,E2 90.0723} C_DIS
LIN {X 1.7174,Y 4.4929,Z 52,A -2.3913,B 0,C 0,E1 0.1598,E2 90.0723} C_DIS
LIN {X 1.0878,Y 4.6871,Z 52,A -2.4062,B 0,C 0,E1 0.1598,E2 90.0723} C_DIS
LIN {X 0.4371,Y 4.7913,Z 52,A -2.4258,B 0,C 0,E1 0.1598,E2 90.0723} C_DIS
LIN {X -0.2217,Y 4.806,Z 52,A -2.4495,B 0,C 0,E1 0.1598,E2 90.0723} C_DIS
LIN {X -0.876,Y 4.7295,Z 52,A -2.4768,B 0,C 0,E1 0.1598,E2 90.0723} C_DIS
LIN {X -1.5144,Y 4.5657,Z 52,A -2.5073,B 0,C 0,E1 0.1598,E2 90.0723} C_DIS
LIN {X -2.1244,Y 4.3166,Z 52,A -2.5404,B 0,C 0,E1 0.1598,E2 90.0722} C_DIS
LIN {X -2.6949,Y 3.9865,Z 52,A -2.5754,B 0,C 0,E1 0.1598,E2 90.0721} C_DIS
LIN {X -3.2137,Y 3.5802,Z 52,A -2.6117,B 0,C 0,E1 0.1598,E2 90.0721} C_DIS
LIN {X -3.6725,Y 3.1071,Z 52,A -2.6486,B 0,C 0,E1 0.1598,E2 90.0719} C_DIS
LIN {X -4.062,Y 2.5757,Z 52,A -2.6855,B 0,C 0,E1 0.1598,E2 90.0719} C_DIS
LIN {X -4.376,Y 1.9966,Z 52,A -2.7216,B 0,C 0,E1 0.1598,E2 90.0718} C_DIS
LIN {X -4.6076,Y 1.3798,Z 52,A -2.7563,B 0,C 0,E1 0.1598,E2 90.0717} C_DIS
LIN {X -4.7528,Y 0.7372,Z 52,A -2.7889,B 0,C 0,E1 0.1598,E2 90.0717} C_DIS
LIN {X -4.8081,Y 0.0808,Z 52,A -2.8187,B 0,C 0,E1 0.1598,E2 90.0716} C_DIS
LIN {X -4.7765,Y -0.5772,Z 52,A -2.8455,B 0,C 0,E1 0.1598,E2 90.0716} C_DIS
LIN {X -4.6504,Y -1.2239,Z 52,A -2.8683,B 0,C 0,E1 0.1598,E2 90.0716} C_DIS
LIN {X -4.4403,Y -1.8483,Z 52,A -2.8871,B 0,C 0,E1 0.1598,E2 90.0716} C_DIS
LIN {X -4.1464,Y -2.438,Z 52,A -2.9014,B 0,C 0,E1 0.1598,E2 90.0716} C_DIS
LIN {X -3.7737,Y -2.9815,Z 52,A -2.9108,B 0,C 0,E1 0.1598,E2 90.0716} C_DIS
LIN {X -3.3306,Y -3.4689,Z 52,A -2.9153,B 0,C 0,E1 0.1598,E2 90.0716} C_DIS
LIN {X -2.8246,Y -3.8908,Z 52,A -2.9147,B 0,C 0,E1 0.1598,E2 90.0716} C_DIS
LIN {X -1.9302,Y -4.4107,Z 52,A -2.9039,B 0,C 0,E1 0.1598,E2 90.0716} C_DIS
LIN {X -1.2598,Y -4.6424,Z 52,A -2.8893,B 0,C 0,E1 0.1598,E2 90.0716} C_DIS
LIN {X -0.7046,Y -4.759,Z 52,A -2.8739,B 0,C 0,E1 0.1598,E2 90.0717} C_DIS
LIN {X 0.0025,Y -4.8154,Z 52,A -2.8503,B 0,C 0,E1 0.1598,E2 90.0717} C_DIS
Enddeposition()
LIN {X 0.0025,Y -4.8154,Z 52,A -2.8503,B 0,C 0,E1 0.1598,E2 90.0717} C_DIS
Startdeposition()
$VEL.CP = VEL_PRINT
LIN {X -0.5747,Y -5.6832,Z 52,A -100.1251,B 7.4649,C -0.3326,E1 7.4527,E2 186.3358} C_DIS
LIN {X -1.3395,Y -5.5542,Z 52,A -107.9927,B 7.4648,C -0.336,E1 7.4312,E2 194.2067} C_DIS
LIN {X -2.0798,Y -5.3226,Z 52,A -115.9247,B 7.4645,C -0.3425,E1 7.4103,E2 202.1415} C_DIS
LIN {X -2.782,Y -4.9926,Z 52,A -123.783,B 7.464,C -0.3518,E1 7.3908,E2 210.0018} C_DIS
LIN {X -3.7786,Y -4.292,Z 52,A -136.6312,B 7.463,C -0.3724,E1 7.3623,E2 222.8536} C_DIS
LIN {X -4.4842,Y -3.5478,Z 52,A -148.1417,B 7.4619,C -0.3957,E1 7.3414,E2 234.3685} C_DIS
LIN {X -4.9398,Y -2.8844,Z 52,A -157.1619,B 7.4607,C -0.4167,E1 7.3287,E2 243.3911} C_DIS
LIN {X -5.4864,Y -1.6161,Z 52,A -169.1531,B 7.4588,C -0.4491,E1 7.3171,E2 255.3713} C_DIS
LIN {X -5.675,Y -0.665,Z 52,A -178.9758,B 7.4572,C -0.4763,E1 7.3126,E2 265.1903} C_DIS
LIN {X -5.7119,Y 0.1097,Z 52,A 173.0619,B 7.4557,C -0.4986,E1 7.3123,E2 273.1496} C_DIS
LIN {X -5.6445,Y 0.8824,Z 52,A 165.2563,B 7.4542,C -0.5205,E1 7.3149,E2 280.9512} C_DIS
LIN {X -5.4737,Y 1.639,Z 52,A 156.9859,B 7.4526,C -0.5429,E1 7.3208,E2 289.2189} C_DIS
LIN {X -5.1992,Y 2.3644,Z 52,A 149.3969,B 7.4512,C -0.5629,E1 7.3289,E2 296.8024} C_DIS
LIN {X -4.8328,Y 3.0479,Z 52,A 141.3943,B 7.4497,C -0.5824,E1 7.3401,E2 304.8009} C_DIS
LIN {X -4.3767,Y 3.6756,Z 52,A 133.4201,B 7.4483,C -0.6001,E1 7.3538,E2 312.7707} C_DIS
LIN {X -3.838,Y 4.2338,Z 52,A 125.4645,B 7.447,C -0.6157,E1 7.3697,E2 320.7218} C_DIS
LIN {X -3.0696,Y 4.8254,Z 52,A 115.1213,B 7.4456,C -0.6322,E1 7.3933,E2 331.0611} C_DIS
Enddeposition()
END
